LIN {X 0,Y 377.649,Z 370.974,A -85,B 0,C 180,E1 -13185.872,E2 -13185.872} C_VEL
LIN {X 0,Y 374.932,Z 477.201,A -85,B 0,C 180,E1 -13187.993,E2 -13187.993} C_VEL
LIN {X 0,Y 374.183,Z 491.579,A -85,B 0,C 180,E1 -13188.499,E2 -13188.499} C_VEL
LIN {X 0,Y 373.169,Z 505.448,A -85,B 0,C 180,E1 -13189.212,E2 -13189.212} C_VEL
LIN {X 0,Y 372.043,Z 517.617,A -85,B 0,C 180,E1 -13190.04,E2 -13190.04} C_VEL
LIN {X 0,Y 370.513,Z 530.576,A -85,B 0,C 180,E1 -13191.157,E2 -13191.157} C_VEL
LIN {X 0,Y 368.92,Z 542.458,A -85,B 0,C 180,E1 -13192.441,E2 -13192.441} C_VEL
LIN {X 0,Y 367.278,Z 553.835,A -85,B 0,C 180,E1 -13193.957,E2 -13193.957} C_VEL
LIN {X 0,Y 365.706,Z 564.018,A -85,B 0,C 180,E1 -13195.628,E2 -13195.628} C_VEL
LIN {X 0,Y 364.372,Z 572.454,A -85,B 0,C 180,E1 -13197.314,E2 -13197.314} C_VEL
LIN {X 0,Y 363.167,Z 579.995,A -85,B 0,C 180,E1 -13199.149,E2 -13199.149} C_VEL
LIN {X 0,Y 362.222,Z 586.133,A -85,B 0,C 180,E1 -13200.985,E2 -13200.985} C_VEL
LIN {X 0,Y 361.531,Z 591.036,A -85,B 0,C 180,E1 -13202.819,E2 -13202.819} C_VEL
LIN {X 0,Y 361.006,Z 594.853,A -85,B 0,C 180,E1 -13204.642,E2 -13204.642} C_VEL
LIN {X 0,Y 360.671,Z 597.534,A -85,B 0,C 180,E1 -13206.324,E2 -13206.324} C_VEL
LIN {X 0,Y 360.375,Z 599.657,A -85,B 0,C 180,E1 -13208.253,E2 -13208.253} C_VEL
LIN {X 0,Y 360.206,Z 600.871,A -85,B 0,C 180,E1 -13210.63,E2 -13210.63} C_VEL
LIN {X 0,Y 360.181,Z 600.626,A -85,B 0,C 180,E1 -13212.982,E2 -13212.982} C_VEL
LIN {X 0,Y 360.246,Z 598.959,A -85,B 0,C 180,E1 -13215.31,E2 -13215.31} C_VEL
LIN {X 0,Y 360.558,Z 595.855,A -85,B 0,C 180,E1 -13217.62,E2 -13217.62} C_VEL
LIN {X 0,Y 360.942,Z 591.269,A -85,B 0,C 180,E1 -13219.908,E2 -13219.908} C_VEL
LIN {X 0,Y 361.382,Z 586.711,A -85,B 0,C 180,E1 -13221.614,E2 -13221.614} C_VEL
LIN {X 0,Y 362.004,Z 580.162,A -85,B 0,C 180,E1 -13223.592,E2 -13223.592} C_VEL
LIN {X 0,Y 362.969,Z 572.024,A -85,B 0,C 180,E1 -13225.559,E2 -13225.559} C_VEL
LIN {X 0,Y 363.95,Z 563.517,A -85,B 0,C 180,E1 -13227.234,E2 -13227.234} C_VEL
LIN {X 0,Y 365.15,Z 553.229,A -85,B 0,C 180,E1 -13228.898,E2 -13228.898} C_VEL
LIN {X 0,Y 366.336,Z 542.888,A -85,B 0,C 180,E1 -13230.276,E2 -13230.276} C_VEL
LIN {X 0,Y 367.487,Z 531.674,A -85,B 0,C 180,E1 -13231.508,E2 -13231.508} C_VEL
LIN {X 0,Y 368.688,Z 519.413,A -85,B 0,C 180,E1 -13232.596,E2 -13232.596} C_VEL
LIN {X 0,Y 369.825,Z 505.784,A -85,B 0,C 180,E1 -13233.542,E2 -13233.542} C_VEL
LIN {X 0,Y 370.628,Z 491.571,A -85,B 0,C 180,E1 -13234.283,E2 -13234.283} C_VEL
LIN {X 0,Y 371.199,Z 477.507,A -85,B 0,C 180,E1 -13234.786,E2 -13234.786} C_VEL
LIN {X 0,Y 371.887,Z 446.589,A -85,B 0,C 180,E1 -13235.423,E2 -13235.423} C_VEL
LIN {X 0,Y 372.953,Z 396.239,A -85,B 0,C 180,E1 -13236.396,E2 -13236.396} C_VEL
LIN {X 0,Y 372.665,Z 390.402,A -85,B 0,C 180,E1 -13236.533,E2 -13236.533} C_VEL
LIN {X 0,Y 370.599,Z 380.961,A -85,B 0,C 180,E1 -13236.854,E2 -13236.854} C_VEL
LIN {X 0,Y 365.85,Z 366.146,A -85,B 0,C 180,E1 -13237.461,E2 -13237.461} C_VEL
LIN {X 0,Y 357.086,Z 342.727,A -85,B 0,C 180,E1 -13238.539,E2 -13238.539} C_VEL
LIN {X 0,Y 356.134,Z 340.083,A -85,B 0,C 180,E1 -13238.698,E2 -13238.698} C_VEL
LIN {X 0,Y 354.975,Z 334.897,A -85,B 0,C 180,E1 -13240.121,E2 -13240.121} C_VEL
LIN {X 0,Y 354.941,Z 334.894,A -85,B 0,C 180,E1 -13244.02,E2 -13244.02} C_VEL
LIN {X 0,Y 354.889,Z 334.9,A -85,B 0,C 180,E1 -13248.093,E2 -13248.093} C_VEL
LIN {X 0,Y 354.816,Z 334.913,A -85,B 0,C 180,E1 -13251.418,E2 -13251.418} C_VEL
LIN {X 0,Y 354.847,Z 334.907,A -85,B 0,C 180,E1 -13254.578,E2 -13254.578} C_VEL
LIN {X 0,Y 354.796,Z 334.913,A -85,B 0,C 180,E1 -13258.387,E2 -13258.387} C_VEL
LIN {X 0,Y 354.778,Z 334.915,A -85,B 0,C 180,E1 -13262.335,E2 -13262.335} C_VEL
LIN {X 0,Y 354.817,Z 334.909,A -85,B 0,C 180,E1 -13265.699,E2 -13265.699} C_VEL
LIN {X 0,Y 354.768,Z 334.916,A -85,B 0,C 180,E1 -13269.413,E2 -13269.413} C_VEL
LIN {X 0,Y 354.78,Z 334.919,A -85,B 0,C 180,E1 -13272.867,E2 -13272.867} C_VEL
LIN {X 0,Y 354.762,Z 334.916,A -85,B 0,C 180,E1 -13276.104,E2 -13276.104} C_VEL
LIN {X 0,Y 354.763,Z 334.917,A -85,B 0,C 180,E1 -13279.176,E2 -13279.176} C_VEL
LIN {X 0,Y 354.799,Z 334.915,A -85,B 0,C 180,E1 -13282.405,E2 -13282.405} C_VEL
LIN {X 0,Y 354.811,Z 334.912,A -85,B 0,C 180,E1 -13284.941,E2 -13284.941} C_VEL
LIN {X 0,Y 354.795,Z 334.917,A -85,B 0,C 180,E1 -13288.406,E2 -13288.406} C_VEL
LIN {X 0,Y 354.798,Z 334.911,A -85,B 0,C 180,E1 -13291.615,E2 -13291.615} C_VEL
LIN {X 0,Y 354.803,Z 334.911,A -85,B 0,C 180,E1 -13295.42,E2 -13295.42} C_VEL
LIN {X 0,Y 354.824,Z 334.908,A -85,B 0,C 180,E1 -13299.113,E2 -13299.113} C_VEL
LIN {X 0,Y 354.862,Z 334.905,A -85,B 0,C 180,E1 -13302.719,E2 -13302.719} C_VEL
LIN {X 0,Y 354.942,Z 334.899,A -85,B 0,C 180,E1 -13306.255,E2 -13306.255} C_VEL
LIN {X 0,Y 354.959,Z 334.893,A -85,B 0,C 180,E1 -13309.736,E2 -13309.736} C_VEL
LIN {X 0,Y 355.093,Z 334.875,A -85,B 0,C 180,E1 -13313.18,E2 -13313.18} C_VEL
LIN {X 0,Y 355.238,Z 334.86,A -85,B 0,C 180,E1 -13317.733,E2 -13317.733} C_VEL
LIN {X 0,Y 355.334,Z 334.85,A -85,B 0,C 180,E1 -13320,E2 -13320} C_VEL
LIN {X 0,Y 355.236,Z 334.86,A -85,B 0,C 180,E1 -13322.268,E2 -13322.268} C_VEL
LIN {X 0,Y 355.107,Z 334.873,A -85,B 0,C 180,E1 -13326.82,E2 -13326.82} C_VEL
LIN {X 0,Y 354.961,Z 334.893,A -85,B 0,C 180,E1 -13330.265,E2 -13330.265} C_VEL
LIN {X 0,Y 354.947,Z 334.896,A -85,B 0,C 180,E1 -13334.019,E2 -13334.019} C_VEL
LIN {X 0,Y 354.927,Z 334.897,A -85,B 0,C 180,E1 -13338.108,E2 -13338.108} C_VEL
LIN {X 0,Y 354.84,Z 334.908,A -85,B 0,C 180,E1 -13342.106,E2 -13342.106} C_VEL
LIN {X 0,Y 354.904,Z 334.902,A -85,B 0,C 180,E1 -13345.827,E2 -13345.827} C_VEL
LIN {X 0,Y 354.822,Z 334.913,A -85,B 0,C 180,E1 -13349.682,E2 -13349.682} C_VEL
LIN {X 0,Y 354.811,Z 334.913,A -85,B 0,C 180,E1 -13353.702,E2 -13353.702} C_VEL
LIN {X 0,Y 354.804,Z 334.911,A -85,B 0,C 180,E1 -13356.459,E2 -13356.459} C_VEL
LIN {X 0,Y 354.829,Z 334.913,A -85,B 0,C 180,E1 -13359.423,E2 -13359.423} C_VEL
LIN {X 0,Y 354.793,Z 334.914,A -85,B 0,C 180,E1 -13362.867,E2 -13362.867} C_VEL
LIN {X 0,Y 354.785,Z 334.913,A -85,B 0,C 180,E1 -13366.105,E2 -13366.105} C_VEL
LIN {X 0,Y 354.792,Z 334.918,A -85,B 0,C 180,E1 -13369.179,E2 -13369.179} C_VEL
LIN {X 0,Y 354.812,Z 334.91,A -85,B 0,C 180,E1 -13372.402,E2 -13372.402} C_VEL
LIN {X 0,Y 354.817,Z 334.914,A -85,B 0,C 180,E1 -13374.94,E2 -13374.94} C_VEL
LIN {X 0,Y 354.837,Z 334.945,A -85,B 0,C 180,E1 -13376.87,E2 -13376.87} C_VEL
LIN {X 0,Y 357.871,Z 348.237,A -85,B 0,C 180,E1 -13380.042,E2 -13380.042} C_VEL
LIN {X 0,Y 360.045,Z 358.455,A -85,B 0,C 180,E1 -13382.38,E2 -13382.38} C_VEL
LIN {X 0,Y 360.126,Z 361.424,A -85,B 0,C 180,E1 -13383.016,E2 -13383.016} C_VEL
LIN {X 0,Y 359.846,Z 364.189,A -85,B 0,C 180,E1 -13383.584,E2 -13383.584} C_VEL
LIN {X 0,Y 366.367,Z 404.572,A -85,B 0,C 180,E1 -13384.865,E2 -13384.865} C_VEL
LIN {X 0,Y 364.3,Z 502.303,A -85,B 0,C 180,E1 -13386.816,E2 -13386.816} C_VEL
LIN {X 0,Y 363.56,Z 517.056,A -85,B 0,C 180,E1 -13387.33,E2 -13387.33} C_VEL
LIN {X 0,Y 362.525,Z 530.545,A -85,B 0,C 180,E1 -13388.012,E2 -13388.012} C_VEL
LIN {X 0,Y 361.356,Z 543.945,A -85,B 0,C 180,E1 -13388.926,E2 -13388.926} C_VEL
LIN {X 0,Y 360.042,Z 556.534,A -85,B 0,C 180,E1 -13390.025,E2 -13390.025} C_VEL
LIN {X 0,Y 358.731,Z 568.174,A -85,B 0,C 180,E1 -13391.287,E2 -13391.287} C_VEL
LIN {X 0,Y 357.614,Z 577.86,A -85,B 0,C 180,E1 -13392.56,E2 -13392.56} C_VEL
LIN {X 0,Y 356.296,Z 588.612,A -85,B 0,C 180,E1 -13394.262,E2 -13394.262} C_VEL
LIN {X 0,Y 355.379,Z 596.927,A -85,B 0,C 180,E1 -13395.862,E2 -13395.862} C_VEL
LIN {X 0,Y 354.607,Z 604.84,A -85,B 0,C 180,E1 -13397.698,E2 -13397.698} C_VEL
LIN {X 0,Y 353.853,Z 611.86,A -85,B 0,C 180,E1 -13399.702,E2 -13399.702} C_VEL
LIN {X 0,Y 353.555,Z 616.713,A -85,B 0,C 180,E1 -13401.425,E2 -13401.425} C_VEL
LIN {X 0,Y 353.386,Z 620.636,A -85,B 0,C 180,E1 -13403.146,E2 -13403.146} C_VEL
LIN {X 0,Y 353.267,Z 624.452,A -85,B 0,C 180,E1 -13405.435,E2 -13405.435} C_VEL
LIN {X 0,Y 353.239,Z 626.831,A -85,B 0,C 180,E1 -13407.718,E2 -13407.718} C_VEL
LIN {X 0,Y 353.329,Z 627.841,A -85,B 0,C 180,E1 -13409.999,E2 -13409.999} C_VEL
LIN {X 0,Y 353.202,Z 627.494,A -85,B 0,C 180,E1 -13412.28,E2 -13412.28} C_VEL
LIN {X 0,Y 353.247,Z 625.81,A -85,B 0,C 180,E1 -13414.563,E2 -13414.563} C_VEL
LIN {X 0,Y 353.395,Z 622.758,A -85,B 0,C 180,E1 -13416.852,E2 -13416.852} C_VEL
LIN {X 0,Y 353.692,Z 618.263,A -85,B 0,C 180,E1 -13419.146,E2 -13419.146} C_VEL
LIN {X 0,Y 354.128,Z 613.835,A -85,B 0,C 180,E1 -13420.866,E2 -13420.866} C_VEL
LIN {X 0,Y 355.078,Z 607.458,A -85,B 0,C 180,E1 -13422.865,E2 -13422.865} C_VEL
LIN {X 0,Y 356.089,Z 599.558,A -85,B 0,C 180,E1 -13424.866,E2 -13424.866} C_VEL
LIN {X 0,Y 357.377,Z 591.334,A -85,B 0,C 180,E1 -13426.567,E2 -13426.567} C_VEL
LIN {X 0,Y 359,Z 581.461,A -85,B 0,C 180,E1 -13428.253,E2 -13428.253} C_VEL
LIN {X 0,Y 360.756,Z 570.523,A -85,B 0,C 180,E1 -13429.784,E2 -13429.784} C_VEL
LIN {X 0,Y 362.6,Z 558.411,A -85,B 0,C 180,E1 -13431.16,E2 -13431.16} C_VEL
LIN {X 0,Y 364.157,Z 546.5,A -85,B 0,C 180,E1 -13432.255,E2 -13432.255} C_VEL
LIN {X 0,Y 365.623,Z 533.389,A -85,B 0,C 180,E1 -13433.205,E2 -13433.205} C_VEL
LIN {X 0,Y 367.002,Z 519.12,A -85,B 0,C 180,E1 -13433.973,E2 -13433.973} C_VEL
LIN {X 0,Y 368.077,Z 504.919,A -85,B 0,C 180,E1 -13434.499,E2 -13434.499} C_VEL
LIN {X 0,Y 368.736,Z 484.2,A -85,B 0,C 180,E1 -13434.97,E2 -13434.97} C_VEL
LIN {X 0,Y 370.703,Z 405.046,A -85,B 0,C 180,E1 -13436.561,E2 -13436.561} C_VEL
LIN {X 0,Y 366.814,Z 382.746,A -85,B 0,C 180,E1 -13437.423,E2 -13437.423} C_VEL
LIN {X 0,Y 363.097,Z 366.604,A -85,B 0,C 180,E1 -13438.154,E2 -13438.154} C_VEL
LIN {X 0,Y 361.741,Z 363.168,A -85,B 0,C 180,E1 -13438.406,E2 -13438.406} C_VEL
LIN {X 0,Y 359.351,Z 352.096,A -85,B 0,C 180,E1 -13441.214,E2 -13441.214} C_VEL
LIN {X 0,Y 356.366,Z 340.467,A -85,B 0,C 180,E1 -13444.383,E2 -13444.383} C_VEL
LIN {X 0,Y 354.819,Z 334.906,A -85,B 0,C 180,E1 -13446.028,E2 -13446.028} C_VEL
LIN {X 0,Y 354.821,Z 334.908,A -85,B 0,C 180,E1 -13449.422,E2 -13449.422} C_VEL
LIN {X 0,Y 354.8,Z 334.909,A -85,B 0,C 180,E1 -13452.869,E2 -13452.869} C_VEL
LIN {X 0,Y 354.763,Z 334.905,A -85,B 0,C 180,E1 -13456.103,E2 -13456.103} C_VEL
LIN {X 0,Y 354.787,Z 334.909,A -85,B 0,C 180,E1 -13459.178,E2 -13459.178} C_VEL
LIN {X 0,Y 354.807,Z 334.912,A -85,B 0,C 180,E1 -13462.4,E2 -13462.4} C_VEL
LIN {X 0,Y 354.807,Z 334.913,A -85,B 0,C 180,E1 -13464.94,E2 -13464.94} C_VEL
LIN {X 0,Y 354.788,Z 334.917,A -85,B 0,C 180,E1 -13468.404,E2 -13468.404} C_VEL
LIN {X 0,Y 354.848,Z 334.907,A -85,B 0,C 180,E1 -13471.618,E2 -13471.618} C_VEL
LIN {X 0,Y 354.892,Z 334.898,A -85,B 0,C 180,E1 -13474.172,E2 -13474.172} C_VEL
LIN {X 0,Y 354.825,Z 334.905,A -85,B 0,C 180,E1 -13477.893,E2 -13477.893} C_VEL
LIN {X 0,Y 354.915,Z 334.895,A -85,B 0,C 180,E1 -13481.891,E2 -13481.891} C_VEL
LIN {X 0,Y 354.935,Z 334.894,A -85,B 0,C 180,E1 -13485.98,E2 -13485.98} C_VEL
LIN {X 0,Y 354.969,Z 334.887,A -85,B 0,C 180,E1 -13489.735,E2 -13489.735} C_VEL
LIN {X 0,Y 355.105,Z 334.872,A -85,B 0,C 180,E1 -13492.036,E2 -13492.036} C_VEL
LIN {X 0,Y 355.079,Z 334.88,A -85,B 0,C 180,E1 -13494.32,E2 -13494.32} C_VEL
LIN {X 0,Y 355.221,Z 334.856,A -85,B 0,C 180,E1 -13497.732,E2 -13497.732} C_VEL
LIN {X 0,Y 355.136,Z 334.866,A -85,B 0,C 180,E1 -13501.134,E2 -13501.134} C_VEL
LIN {X 0,Y 355.223,Z 334.861,A -85,B 0,C 180,E1 -13502.267,E2 -13502.267} C_VEL
LIN {X 0,Y 355.073,Z 334.879,A -85,B 0,C 180,E1 -13506.82,E2 -13506.82} C_VEL
LIN {X 0,Y 354.944,Z 334.896,A -85,B 0,C 180,E1 -13510.265,E2 -13510.265} C_VEL
LIN {X 0,Y 354.933,Z 334.898,A -85,B 0,C 180,E1 -13514.018,E2 -13514.018} C_VEL
LIN {X 0,Y 354.88,Z 334.903,A -85,B 0,C 180,E1 -13518.092,E2 -13518.092} C_VEL
LIN {X 0,Y 354.806,Z 334.908,A -85,B 0,C 180,E1 -13522.107,E2 -13522.107} C_VEL
LIN {X 0,Y 354.839,Z 334.909,A -85,B 0,C 180,E1 -13524.577,E2 -13524.577} C_VEL
LIN {X 0,Y 354.79,Z 334.902,A -85,B 0,C 180,E1 -13528.386,E2 -13528.386} C_VEL
LIN {X 0,Y 354.778,Z 334.913,A -85,B 0,C 180,E1 -13532.334,E2 -13532.334} C_VEL
LIN {X 0,Y 354.813,Z 334.914,A -85,B 0,C 180,E1 -13535.7,E2 -13535.7} C_VEL
LIN {X 0,Y 354.816,Z 334.906,A -85,B 0,C 180,E1 -13539.424,E2 -13539.424} C_VEL
LIN {X 0,Y 354.803,Z 335.09,A -85,B 0,C 180,E1 -13541.176,E2 -13541.176} C_VEL
LIN {X 0,Y 356.505,Z 341.345,A -85,B 0,C 180,E1 -13543.134,E2 -13543.134} C_VEL
LIN {X 0,Y 366.3,Z 360.999,A -85,B 0,C 180,E1 -13544.598,E2 -13544.598} C_VEL
LIN {X 0,Y 371.482,Z 372.961,A -85,B 0,C 180,E1 -13545.359,E2 -13545.359} C_VEL
LIN {X 0,Y 368.723,Z 476.994,A -85,B 0,C 180,E1 -13547.466,E2 -13547.466} C_VEL
LIN {X 0,Y 367.99,Z 491.14,A -85,B 0,C 180,E1 -13547.963,E2 -13547.963} C_VEL
LIN {X 0,Y 366.946,Z 504.304,A -85,B 0,C 180,E1 -13548.628,E2 -13548.628} C_VEL
LIN {X 0,Y 365.644,Z 517.9,A -85,B 0,C 180,E1 -13549.558,E2 -13549.558} C_VEL
LIN {X 0,Y 364.099,Z 530.421,A -85,B 0,C 180,E1 -13550.65,E2 -13550.65} C_VEL
LIN {X 0,Y 362.576,Z 541.429,A -85,B 0,C 180,E1 -13551.843,E2 -13551.843} C_VEL
LIN {X 0,Y 360.792,Z 553.001,A -85,B 0,C 180,E1 -13553.378,E2 -13553.378} C_VEL
LIN {X 0,Y 359.121,Z 563.612,A -85,B 0,C 180,E1 -13555.117,E2 -13555.117} C_VEL
LIN {X 0,Y 357.576,Z 572.703,A -85,B 0,C 180,E1 -13556.949,E2 -13556.949} C_VEL
LIN {X 0,Y 356.31,Z 580.25,A -85,B 0,C 180,E1 -13558.819,E2 -13558.819} C_VEL
LIN {X 0,Y 355.391,Z 585.721,A -85,B 0,C 180,E1 -13560.471,E2 -13560.471} C_VEL
LIN {X 0,Y 354.648,Z 590.535,A -85,B 0,C 180,E1 -13562.246,E2 -13562.246} C_VEL
LIN {X 0,Y 353.9,Z 595.679,A -85,B 0,C 180,E1 -13564.726,E2 -13564.726} C_VEL
LIN {X 0,Y 353.531,Z 598.345,A -85,B 0,C 180,E1 -13566.574,E2 -13566.574} C_VEL
LIN {X 0,Y 353.205,Z 600.546,A -85,B 0,C 180,E1 -13569.014,E2 -13569.014} C_VEL
LIN {X 0,Y 353.083,Z 601.243,A -85,B 0,C 180,E1 -13571.431,E2 -13571.431} C_VEL
LIN {X 0,Y 353.113,Z 600.455,A -85,B 0,C 180,E1 -13573.822,E2 -13573.822} C_VEL
LIN {X 0,Y 353.218,Z 598.249,A -85,B 0,C 180,E1 -13576.188,E2 -13576.188} C_VEL
LIN {X 0,Y 353.507,Z 595.671,A -85,B 0,C 180,E1 -13577.952,E2 -13577.952} C_VEL
LIN {X 0,Y 353.802,Z 592.19,A -85,B 0,C 180,E1 -13579.703,E2 -13579.703} C_VEL
LIN {X 0,Y 354.242,Z 587.817,A -85,B 0,C 180,E1 -13581.444,E2 -13581.444} C_VEL
LIN {X 0,Y 354.882,Z 581.464,A -85,B 0,C 180,E1 -13583.463,E2 -13583.463} C_VEL
LIN {X 0,Y 355.821,Z 573.552,A -85,B 0,C 180,E1 -13585.47,E2 -13585.47} C_VEL
LIN {X 0,Y 356.793,Z 565.299,A -85,B 0,C 180,E1 -13587.178,E2 -13587.178} C_VEL
LIN {X 0,Y 358.063,Z 555.338,A -85,B 0,C 180,E1 -13588.876,E2 -13588.876} C_VEL
LIN {X 0,Y 359.377,Z 544.282,A -85,B 0,C 180,E1 -13590.421,E2 -13590.421} C_VEL
LIN {X 0,Y 360.536,Z 533.314,A -85,B 0,C 180,E1 -13591.677,E2 -13591.677} C_VEL
LIN {X 0,Y 361.767,Z 521.402,A -85,B 0,C 180,E1 -13592.785,E2 -13592.785} C_VEL
LIN {X 0,Y 362.933,Z 508.295,A -85,B 0,C 180,E1 -13593.748,E2 -13593.748} C_VEL
LIN {X 0,Y 363.798,Z 494.108,A -85,B 0,C 180,E1 -13594.537,E2 -13594.537} C_VEL
LIN {X 0,Y 364.424,Z 481.109,A -85,B 0,C 180,E1 -13595.049,E2 -13595.049} C_VEL
LIN {X 0,Y 364.92,Z 464.085,A -85,B 0,C 180,E1 -13595.458,E2 -13595.458} C_VEL
LIN {X 0,Y 366.898,Z 370.233,A -85,B 0,C 180,E1 -13597.308,E2 -13597.308} C_VEL
LIN {X 0,Y 365.85,Z 366.146,A -85,B 0,C 180,E1 -13597.461,E2 -13597.461} C_VEL
LIN {X 0,Y 363.54,Z 360.985,A -85,B 0,C 180,E1 -13597.72,E2 -13597.72} C_VEL
LIN {X 0,Y 360.254,Z 356.432,A -85,B 0,C 180,E1 -13598.032,E2 -13598.032} C_VEL
LIN {X 0,Y 351.868,Z 346.34,A -85,B 0,C 180,E1 -13598.818,E2 -13598.818} C_VEL
LIN {X 0,Y 349.207,Z 341.334,A -85,B 0,C 180,E1 -13599.117,E2 -13599.117} C_VEL
LIN {X 0,Y 348.965,Z 340.469,A -85,B 0,C 180,E1 -13599.161,E2 -13599.161} C_VEL
LIN {X 0,Y 347.894,Z 335.778,A -85,B 0,C 180,E1 -13600.476,E2 -13600.476} C_VEL
LIN {X 0,Y 347.897,Z 335.772,A -85,B 0,C 180,E1 -13604.151,E2 -13604.151} C_VEL
LIN {X 0,Y 347.828,Z 335.78,A -85,B 0,C 180,E1 -13608.26,E2 -13608.26} C_VEL
LIN {X 0,Y 347.763,Z 335.79,A -85,B 0,C 180,E1 -13611.626,E2 -13611.626} C_VEL
LIN {X 0,Y 347.766,Z 335.794,A -85,B 0,C 180,E1 -13615.113,E2 -13615.113} C_VEL
LIN {X 0,Y 347.743,Z 335.796,A -85,B 0,C 180,E1 -13619.017,E2 -13619.017} C_VEL
LIN {X 0,Y 347.73,Z 335.797,A -85,B 0,C 180,E1 -13623.073,E2 -13623.073} C_VEL
LIN {X 0,Y 347.765,Z 335.787,A -85,B 0,C 180,E1 -13626.065,E2 -13626.065} C_VEL
LIN {X 0,Y 347.73,Z 335.797,A -85,B 0,C 180,E1 -13628.796,E2 -13628.796} C_VEL
LIN {X 0,Y 347.739,Z 335.79,A -85,B 0,C 180,E1 -13631.833,E2 -13631.833} C_VEL
LIN {X 0,Y 347.7,Z 335.798,A -85,B 0,C 180,E1 -13635.029,E2 -13635.029} C_VEL
LIN {X 0,Y 347.738,Z 335.794,A -85,B 0,C 180,E1 -13638.401,E2 -13638.401} C_VEL
LIN {X 0,Y 347.762,Z 335.788,A -85,B 0,C 180,E1 -13642.015,E2 -13642.015} C_VEL
LIN {X 0,Y 347.745,Z 335.789,A -85,B 0,C 180,E1 -13645.537,E2 -13645.537} C_VEL
LIN {X 0,Y 347.746,Z 335.793,A -85,B 0,C 180,E1 -13648.301,E2 -13648.301} C_VEL
LIN {X 0,Y 347.745,Z 335.791,A -85,B 0,C 180,E1 -13650.985,E2 -13650.985} C_VEL
LIN {X 0,Y 347.734,Z 335.791,A -85,B 0,C 180,E1 -13653.6,E2 -13653.6} C_VEL
LIN {X 0,Y 347.75,Z 335.793,A -85,B 0,C 180,E1 -13656.16,E2 -13656.16} C_VEL
LIN {X 0,Y 347.778,Z 335.788,A -85,B 0,C 180,E1 -13659.908,E2 -13659.908} C_VEL
LIN {X 0,Y 347.803,Z 335.783,A -85,B 0,C 180,E1 -13663.567,E2 -13663.567} C_VEL
LIN {X 0,Y 347.89,Z 335.769,A -85,B 0,C 180,E1 -13667.161,E2 -13667.161} C_VEL
LIN {X 0,Y 347.938,Z 335.767,A -85,B 0,C 180,E1 -13670.701,E2 -13670.701} C_VEL
LIN {X 0,Y 348.047,Z 335.757,A -85,B 0,C 180,E1 -13674.206,E2 -13674.206} C_VEL
LIN {X 0,Y 348.199,Z 335.735,A -85,B 0,C 180,E1 -13677.687,E2 -13677.687} C_VEL
LIN {X 0,Y 348.286,Z 335.726,A -85,B 0,C 180,E1 -13680,E2 -13680} C_VEL
LIN {X 0,Y 348.198,Z 335.736,A -85,B 0,C 180,E1 -13682.314,E2 -13682.314} C_VEL
LIN {X 0,Y 348.074,Z 335.749,A -85,B 0,C 180,E1 -13686.959,E2 -13686.959} C_VEL
LIN {X 0,Y 347.901,Z 335.771,A -85,B 0,C 180,E1 -13690.476,E2 -13690.476} C_VEL
LIN {X 0,Y 347.903,Z 335.772,A -85,B 0,C 180,E1 -13694.15,E2 -13694.15} C_VEL
LIN {X 0,Y 347.895,Z 335.772,A -85,B 0,C 180,E1 -13698.29,E2 -13698.29} C_VEL
LIN {X 0,Y 347.795,Z 335.79,A -85,B 0,C 180,E1 -13701.636,E2 -13701.636} C_VEL
LIN {X 0,Y 347.817,Z 335.782,A -85,B 0,C 180,E1 -13705.108,E2 -13705.108} C_VEL
LIN {X 0,Y 347.813,Z 335.786,A -85,B 0,C 180,E1 -13707.694,E2 -13707.694} C_VEL
LIN {X 0,Y 347.754,Z 335.789,A -85,B 0,C 180,E1 -13710.348,E2 -13710.348} C_VEL
LIN {X 0,Y 347.753,Z 335.79,A -85,B 0,C 180,E1 -13714.044,E2 -13714.044} C_VEL
LIN {X 0,Y 347.769,Z 335.793,A -85,B 0,C 180,E1 -13717.32,E2 -13717.32} C_VEL
LIN {X 0,Y 347.737,Z 335.791,A -85,B 0,C 180,E1 -13720.297,E2 -13720.297} C_VEL
LIN {X 0,Y 347.728,Z 335.797,A -85,B 0,C 180,E1 -13723.408,E2 -13723.408} C_VEL
LIN {X 0,Y 347.732,Z 335.793,A -85,B 0,C 180,E1 -13726.685,E2 -13726.685} C_VEL
LIN {X 0,Y 347.751,Z 335.79,A -85,B 0,C 180,E1 -13730.173,E2 -13730.173} C_VEL
LIN {X 0,Y 347.766,Z 335.79,A -85,B 0,C 180,E1 -13732.679,E2 -13732.679} C_VEL
LIN {X 0,Y 347.787,Z 335.786,A -85,B 0,C 180,E1 -13736.445,E2 -13736.445} C_VEL
LIN {X 0,Y 351.046,Z 350.09,A -85,B 0,C 180,E1 -13739.966,E2 -13739.966} C_VEL
LIN {X 0,Y 353.233,Z 360.748,A -85,B 0,C 180,E1 -13742.445,E2 -13742.445} C_VEL
LIN {X 0,Y 353.094,Z 363.95,A -85,B 0,C 180,E1 -13743.127,E2 -13743.127} C_VEL
LIN {X 0,Y 359.723,Z 405.351,A -85,B 0,C 180,E1 -13744.469,E2 -13744.469} C_VEL
LIN {X 0,Y 357.635,Z 502.009,A -85,B 0,C 180,E1 -13746.435,E2 -13746.435} C_VEL
LIN {X 0,Y 356.868,Z 516.772,A -85,B 0,C 180,E1 -13746.957,E2 -13746.957} C_VEL
LIN {X 0,Y 355.807,Z 530.266,A -85,B 0,C 180,E1 -13747.651,E2 -13747.651} C_VEL
LIN {X 0,Y 354.558,Z 543.932,A -85,B 0,C 180,E1 -13748.602,E2 -13748.602} C_VEL
LIN {X 0,Y 353.335,Z 555.54,A -85,B 0,C 180,E1 -13749.629,E2 -13749.629} C_VEL
LIN {X 0,Y 351.911,Z 567.301,A -85,B 0,C 180,E1 -13750.911,E2 -13750.911} C_VEL
LIN {X 0,Y 350.741,Z 577.088,A -85,B 0,C 180,E1 -13752.206,E2 -13752.206} C_VEL
LIN {X 0,Y 349.393,Z 587.927,A -85,B 0,C 180,E1 -13753.943,E2 -13753.943} C_VEL
LIN {X 0,Y 348.32,Z 597.086,A -85,B 0,C 180,E1 -13755.737,E2 -13755.737} C_VEL
LIN {X 0,Y 347.485,Z 605.424,A -85,B 0,C 180,E1 -13757.738,E2 -13757.738} C_VEL
LIN {X 0,Y 346.807,Z 611.367,A -85,B 0,C 180,E1 -13759.49,E2 -13759.49} C_VEL
LIN {X 0,Y 346.486,Z 616.271,A -85,B 0,C 180,E1 -13761.249,E2 -13761.249} C_VEL
LIN {X 0,Y 346.308,Z 620.24,A -85,B 0,C 180,E1 -13763.005,E2 -13763.005} C_VEL
LIN {X 0,Y 346.186,Z 624.099,A -85,B 0,C 180,E1 -13765.341,E2 -13765.341} C_VEL
LIN {X 0,Y 346.145,Z 626.515,A -85,B 0,C 180,E1 -13767.672,E2 -13767.672} C_VEL
LIN {X 0,Y 346.234,Z 627.562,A -85,B 0,C 180,E1 -13769.999,E2 -13769.999} C_VEL
LIN {X 0,Y 346.111,Z 627.252,A -85,B 0,C 180,E1 -13772.326,E2 -13772.326} C_VEL
LIN {X 0,Y 346.146,Z 625.607,A -85,B 0,C 180,E1 -13774.657,E2 -13774.657} C_VEL
LIN {X 0,Y 346.32,Z 622.596,A -85,B 0,C 180,E1 -13776.993,E2 -13776.993} C_VEL
LIN {X 0,Y 346.648,Z 618.142,A -85,B 0,C 180,E1 -13779.333,E2 -13779.333} C_VEL
LIN {X 0,Y 347.352,Z 612.126,A -85,B 0,C 180,E1 -13781.672,E2 -13781.672} C_VEL
LIN {X 0,Y 348.334,Z 605.389,A -85,B 0,C 180,E1 -13783.712,E2 -13783.712} C_VEL
LIN {X 0,Y 349.635,Z 597.041,A -85,B 0,C 180,E1 -13785.744,E2 -13785.744} C_VEL
LIN {X 0,Y 351.077,Z 588.387,A -85,B 0,C 180,E1 -13787.473,E2 -13787.473} C_VEL
LIN {X 0,Y 352.891,Z 577.94,A -85,B 0,C 180,E1 -13789.183,E2 -13789.183} C_VEL
LIN {X 0,Y 354.809,Z 566.292,A -85,B 0,C 180,E1 -13790.735,E2 -13790.735} C_VEL
LIN {X 0,Y 356.549,Z 554.676,A -85,B 0,C 180,E1 -13791.993,E2 -13791.993} C_VEL
LIN {X 0,Y 358.248,Z 541.93,A -85,B 0,C 180,E1 -13793.1,E2 -13793.1} C_VEL
LIN {X 0,Y 359.782,Z 528.732,A -85,B 0,C 180,E1 -13793.987,E2 -13793.987} C_VEL
LIN {X 0,Y 361.083,Z 515.203,A -85,B 0,C 180,E1 -13794.66,E2 -13794.66} C_VEL
LIN {X 0,Y 362.01,Z 501.478,A -85,B 0,C 180,E1 -13795.129,E2 -13795.129} C_VEL
LIN {X 0,Y 364.561,Z 406.286,A -85,B 0,C 180,E1 -13797.095,E2 -13797.095} C_VEL
LIN {X 0,Y 360.933,Z 384.935,A -85,B 0,C 180,E1 -13797.94,E2 -13797.94} C_VEL
LIN {X 0,Y 357.328,Z 369.42,A -85,B 0,C 180,E1 -13798.672,E2 -13798.672} C_VEL
LIN {X 0,Y 354.555,Z 362.91,A -85,B 0,C 180,E1 -13799.139,E2 -13799.139} C_VEL
LIN {X 0,Y 351.838,Z 350.947,A -85,B 0,C 180,E1 -13802.297,E2 -13802.297} C_VEL
LIN {X 0,Y 349.331,Z 341.44,A -85,B 0,C 180,E1 -13804.993,E2 -13804.993} C_VEL
LIN {X 0,Y 347.772,Z 335.786,A -85,B 0,C 180,E1 -13806.724,E2 -13806.724} C_VEL
LIN {X 0,Y 347.752,Z 335.796,A -85,B 0,C 180,E1 -13810.293,E2 -13810.293} C_VEL
LIN {X 0,Y 347.74,Z 335.796,A -85,B 0,C 180,E1 -13813.404,E2 -13813.404} C_VEL
LIN {X 0,Y 347.721,Z 335.786,A -85,B 0,C 180,E1 -13816.685,E2 -13816.685} C_VEL
LIN {X 0,Y 347.743,Z 335.776,A -85,B 0,C 180,E1 -13820.172,E2 -13820.172} C_VEL
LIN {X 0,Y 347.76,Z 335.794,A -85,B 0,C 180,E1 -13822.679,E2 -13822.679} C_VEL
LIN {X 0,Y 347.742,Z 335.795,A -85,B 0,C 180,E1 -13825.955,E2 -13825.955} C_VEL
LIN {X 0,Y 347.758,Z 335.79,A -85,B 0,C 180,E1 -13829.653,E2 -13829.653} C_VEL
LIN {X 0,Y 347.846,Z 335.777,A -85,B 0,C 180,E1 -13832.743,E2 -13832.743} C_VEL
LIN {X 0,Y 347.779,Z 335.787,A -85,B 0,C 180,E1 -13836.161,E2 -13836.161} C_VEL
LIN {X 0,Y 347.805,Z 335.784,A -85,B 0,C 180,E1 -13839.909,E2 -13839.909} C_VEL
LIN {X 0,Y 347.859,Z 335.78,A -85,B 0,C 180,E1 -13842.359,E2 -13842.359} C_VEL
LIN {X 0,Y 347.89,Z 335.771,A -85,B 0,C 180,E1 -13845.97,E2 -13845.97} C_VEL
LIN {X 0,Y 347.92,Z 335.763,A -85,B 0,C 180,E1 -13849.525,E2 -13849.525} C_VEL
LIN {X 0,Y 348.065,Z 335.751,A -85,B 0,C 180,E1 -13851.874,E2 -13851.874} C_VEL
LIN {X 0,Y 348.055,Z 335.753,A -85,B 0,C 180,E1 -13854.205,E2 -13854.205} C_VEL
LIN {X 0,Y 348.183,Z 335.732,A -85,B 0,C 180,E1 -13857.686,E2 -13857.686} C_VEL
LIN {X 0,Y 348.107,Z 335.741,A -85,B 0,C 180,E1 -13861.156,E2 -13861.156} C_VEL
LIN {X 0,Y 348.185,Z 335.737,A -85,B 0,C 180,E1 -13862.313,E2 -13862.313} C_VEL
LIN {X 0,Y 348.04,Z 335.755,A -85,B 0,C 180,E1 -13866.959,E2 -13866.959} C_VEL
LIN {X 0,Y 347.884,Z 335.775,A -85,B 0,C 180,E1 -13870.475,E2 -13870.475} C_VEL
LIN {X 0,Y 347.89,Z 335.775,A -85,B 0,C 180,E1 -13874.15,E2 -13874.15} C_VEL
LIN {X 0,Y 347.819,Z 335.783,A -85,B 0,C 180,E1 -13878.259,E2 -13878.259} C_VEL
LIN {X 0,Y 347.758,Z 335.788,A -85,B 0,C 180,E1 -13881.626,E2 -13881.626} C_VEL
LIN {X 0,Y 347.759,Z 335.79,A -85,B 0,C 180,E1 -13885.112,E2 -13885.112} C_VEL
LIN {X 0,Y 347.727,Z 335.787,A -85,B 0,C 180,E1 -13887.701,E2 -13887.701} C_VEL
LIN {X 0,Y 347.732,Z 335.798,A -85,B 0,C 180,E1 -13890.349,E2 -13890.349} C_VEL
LIN {X 0,Y 347.74,Z 335.793,A -85,B 0,C 180,E1 -13894.044,E2 -13894.044} C_VEL
LIN {X 0,Y 347.752,Z 335.789,A -85,B 0,C 180,E1 -13897.321,E2 -13897.321} C_VEL
LIN {X 0,Y 347.757,Z 335.873,A -85,B 0,C 180,E1 -13900.483,E2 -13900.483} C_VEL
LIN {X 0,Y 349.262,Z 341.566,A -85,B 0,C 180,E1 -13902.343,E2 -13902.343} C_VEL
LIN {X 0,Y 359.506,Z 361.601,A -85,B 0,C 180,E1 -13903.934,E2 -13903.934} C_VEL
LIN {X 0,Y 365.379,Z 374.94,A -85,B 0,C 180,E1 -13904.83,E2 -13904.83} C_VEL
LIN {X 0,Y 362.51,Z 477.449,A -85,B 0,C 180,E1 -13906.94,E2 -13906.94} C_VEL
LIN {X 0,Y 361.734,Z 491.51,A -85,B 0,C 180,E1 -13907.442,E2 -13907.442} C_VEL
LIN {X 0,Y 360.65,Z 504.591,A -85,B 0,C 180,E1 -13908.113,E2 -13908.113} C_VEL
LIN {X 0,Y 359.276,Z 518.218,A -85,B 0,C 180,E1 -13909.058,E2 -13909.058} C_VEL
LIN {X 0,Y 357.741,Z 530.294,A -85,B 0,C 180,E1 -13910.126,E2 -13910.126} C_VEL
LIN {X 0,Y 356.075,Z 541.729,A -85,B 0,C 180,E1 -13911.379,E2 -13911.379} C_VEL
LIN {X 0,Y 354.341,Z 552.595,A -85,B 0,C 180,E1 -13912.838,E2 -13912.838} C_VEL
LIN {X 0,Y 352.768,Z 561.938,A -85,B 0,C 180,E1 -13914.359,E2 -13914.359} C_VEL
LIN {X 0,Y 351.063,Z 571.519,A -85,B 0,C 180,E1 -13916.254,E2 -13916.254} C_VEL
LIN {X 0,Y 349.798,Z 578.601,A -85,B 0,C 180,E1 -13917.966,E2 -13917.966} C_VEL
LIN {X 0,Y 348.496,Z 585.888,A -85,B 0,C 180,E1 -13920.13,E2 -13920.13} C_VEL
LIN {X 0,Y 347.574,Z 591.556,A -85,B 0,C 180,E1 -13922.287,E2 -13922.287} C_VEL
LIN {X 0,Y 346.966,Z 595.38,A -85,B 0,C 180,E1 -13924.185,E2 -13924.185} C_VEL
LIN {X 0,Y 346.547,Z 598.232,A -85,B 0,C 180,E1 -13926.073,E2 -13926.073} C_VEL
LIN {X 0,Y 346.151,Z 600.61,A -85,B 0,C 180,E1 -13928.565,E2 -13928.565} C_VEL
LIN {X 0,Y 346.015,Z 601.486,A -85,B 0,C 180,E1 -13931.037,E2 -13931.037} C_VEL
LIN {X 0,Y 346.005,Z 600.913,A -85,B 0,C 180,E1 -13933.48,E2 -13933.48} C_VEL
LIN {X 0,Y 346.117,Z 598.895,A -85,B 0,C 180,E1 -13935.898,E2 -13935.898} C_VEL
LIN {X 0,Y 346.492,Z 595.397,A -85,B 0,C 180,E1 -13938.299,E2 -13938.299} C_VEL
LIN {X 0,Y 346.934,Z 590.391,A -85,B 0,C 180,E1 -13940.675,E2 -13940.675} C_VEL
LIN {X 0,Y 347.547,Z 585.148,A -85,B 0,C 180,E1 -13942.573,E2 -13942.573} C_VEL
LIN {X 0,Y 348.239,Z 578.552,A -85,B 0,C 180,E1 -13944.5,E2 -13944.5} C_VEL
LIN {X 0,Y 349.374,Z 569.87,A -85,B 0,C 180,E1 -13946.541,E2 -13946.541} C_VEL
LIN {X 0,Y 350.543,Z 560.807,A -85,B 0,C 180,E1 -13948.278,E2 -13948.278} C_VEL
LIN {X 0,Y 351.839,Z 549.87,A -85,B 0,C 180,E1 -13950.001,E2 -13950.001} C_VEL
LIN {X 0,Y 353.222,Z 538.706,A -85,B 0,C 180,E1 -13951.426,E2 -13951.426} C_VEL
LIN {X 0,Y 354.517,Z 526.412,A -85,B 0,C 180,E1 -13952.7,E2 -13952.7} C_VEL
LIN {X 0,Y 355.823,Z 512.609,A -85,B 0,C 180,E1 -13953.823,E2 -13953.823} C_VEL
LIN {X 0,Y 356.831,Z 499.154,A -85,B 0,C 180,E1 -13954.661,E2 -13954.661} C_VEL
LIN {X 0,Y 357.57,Z 485.359,A -85,B 0,C 180,E1 -13955.287,E2 -13955.287} C_VEL
LIN {X 0,Y 358.123,Z 472.492,A -85,B 0,C 180,E1 -13955.667,E2 -13955.667} C_VEL
LIN {X 0,Y 360.314,Z 371.491,A -85,B 0,C 180,E1 -13957.704,E2 -13957.704} C_VEL
LIN {X 0,Y 358.222,Z 364.76,A -85,B 0,C 180,E1 -13957.985,E2 -13957.985} C_VEL
LIN {X 0,Y 349.894,Z 342.978,A -85,B 0,C 180,E1 -13959.031,E2 -13959.031} C_VEL
LIN {X 0,Y 349.207,Z 341.334,A -85,B 0,C 180,E1 -13959.117,E2 -13959.117} C_VEL
LIN {X 0,Y 348.09,Z 340.136,A -85,B 0,C 180,E1 -13959.316,E2 -13959.316} C_VEL
LIN {X 0,Y 343.923,Z 337.36,A -85,B 0,C 180,E1 -13960.411,E2 -13960.411} C_VEL
LIN {X 0,Y 341.407,Z 336.789,A -85,B 0,C 180,E1 -13961.523,E2 -13961.523} C_VEL
LIN {X 0,Y 340.83,Z 336.652,A -85,B 0,C 180,E1 -13962.267,E2 -13962.267} C_VEL
LIN {X 0,Y 340.816,Z 336.657,A -85,B 0,C 180,E1 -13965.551,E2 -13965.551} C_VEL
LIN {X 0,Y 340.762,Z 336.666,A -85,B 0,C 180,E1 -13969.269,E2 -13969.269} C_VEL
LIN {X 0,Y 340.705,Z 336.673,A -85,B 0,C 180,E1 -13973.075,E2 -13973.075} C_VEL
LIN {X 0,Y 340.714,Z 336.667,A -85,B 0,C 180,E1 -13975.67,E2 -13975.67} C_VEL
LIN {X 0,Y 340.701,Z 336.668,A -85,B 0,C 180,E1 -13979.676,E2 -13979.676} C_VEL
LIN {X 0,Y 340.68,Z 336.671,A -85,B 0,C 180,E1 -13982.437,E2 -13982.437} C_VEL
LIN {X 0,Y 340.715,Z 336.667,A -85,B 0,C 180,E1 -13985.28,E2 -13985.28} C_VEL
LIN {X 0,Y 340.692,Z 336.669,A -85,B 0,C 180,E1 -13988.383,E2 -13988.383} C_VEL
LIN {X 0,Y 340.69,Z 336.669,A -85,B 0,C 180,E1 -13992.045,E2 -13992.045} C_VEL
LIN {X 0,Y 340.649,Z 336.674,A -85,B 0,C 180,E1 -13996.228,E2 -13996.228} C_VEL
LIN {X 0,Y 340.669,Z 336.677,A -85,B 0,C 180,E1 -13998.689,E2 -13998.689} C_VEL
LIN {X 0,Y 340.718,Z 336.664,A -85,B 0,C 180,E1 -14001.771,E2 -14001.771} C_VEL
LIN {X 0,Y 340.724,Z 336.663,A -85,B 0,C 180,E1 -14005.596,E2 -14005.596} C_VEL
LIN {X 0,Y 340.695,Z 336.67,A -85,B 0,C 180,E1 -14008.956,E2 -14008.956} C_VEL
LIN {X 0,Y 340.711,Z 336.667,A -85,B 0,C 180,E1 -14013.013,E2 -14013.013} C_VEL
LIN {X 0,Y 340.702,Z 336.668,A -85,B 0,C 180,E1 -14016.926,E2 -14016.926} C_VEL
LIN {X 0,Y 340.723,Z 336.667,A -85,B 0,C 180,E1 -14020.73,E2 -14020.73} C_VEL
LIN {X 0,Y 340.796,Z 336.658,A -85,B 0,C 180,E1 -14024.45,E2 -14024.45} C_VEL
LIN {X 0,Y 340.852,Z 336.649,A -85,B 0,C 180,E1 -14028.101,E2 -14028.101} C_VEL
LIN {X 0,Y 340.983,Z 336.634,A -85,B 0,C 180,E1 -14031.705,E2 -14031.705} C_VEL
LIN {X 0,Y 341.021,Z 336.634,A -85,B 0,C 180,E1 -14034.086,E2 -14034.086} C_VEL
LIN {X 0,Y 341.161,Z 336.611,A -85,B 0,C 180,E1 -14037.639,E2 -14037.639} C_VEL
LIN {X 0,Y 341.237,Z 336.602,A -85,B 0,C 180,E1 -14040,E2 -14040} C_VEL
LIN {X 0,Y 341.135,Z 336.615,A -85,B 0,C 180,E1 -14042.362,E2 -14042.362} C_VEL
LIN {X 0,Y 341.022,Z 336.628,A -85,B 0,C 180,E1 -14047.103,E2 -14047.103} C_VEL
LIN {X 0,Y 340.852,Z 336.649,A -85,B 0,C 180,E1 -14050.695,E2 -14050.695} C_VEL
LIN {X 0,Y 340.868,Z 336.647,A -85,B 0,C 180,E1 -14054.325,E2 -14054.325} C_VEL
LIN {X 0,Y 340.842,Z 336.65,A -85,B 0,C 180,E1 -14058.466,E2 -14058.466} C_VEL
LIN {X 0,Y 340.759,Z 336.664,A -85,B 0,C 180,E1 -14061.857,E2 -14061.857} C_VEL
LIN {X 0,Y 340.777,Z 336.663,A -85,B 0,C 180,E1 -14065.664,E2 -14065.664} C_VEL
LIN {X 0,Y 340.733,Z 336.663,A -85,B 0,C 180,E1 -14068.321,E2 -14068.321} C_VEL
LIN {X 0,Y 340.702,Z 336.669,A -85,B 0,C 180,E1 -14071.045,E2 -14071.045} C_VEL
LIN {X 0,Y 340.723,Z 336.67,A -85,B 0,C 180,E1 -14075.279,E2 -14075.279} C_VEL
LIN {X 0,Y 340.716,Z 336.664,A -85,B 0,C 180,E1 -14078.386,E2 -14078.386} C_VEL
LIN {X 0,Y 340.704,Z 336.668,A -85,B 0,C 180,E1 -14082.045,E2 -14082.045} C_VEL
LIN {X 0,Y 340.689,Z 336.673,A -85,B 0,C 180,E1 -14085.461,E2 -14085.461} C_VEL
LIN {X 0,Y 340.69,Z 336.671,A -85,B 0,C 180,E1 -14088.69,E2 -14088.69} C_VEL
LIN {X 0,Y 340.737,Z 336.665,A -85,B 0,C 180,E1 -14091.772,E2 -14091.772} C_VEL
LIN {X 0,Y 340.727,Z 336.667,A -85,B 0,C 180,E1 -14095.595,E2 -14095.595} C_VEL
LIN {X 0,Y 340.712,Z 336.668,A -85,B 0,C 180,E1 -14096.085,E2 -14096.085} C_VEL
LIN {X 0,Y 343.965,Z 350.84,A -85,B 0,C 180,E1 -14099.621,E2 -14099.621} C_VEL
LIN {X 0,Y 346.209,Z 361.512,A -85,B 0,C 180,E1 -14102.166,E2 -14102.166} C_VEL
LIN {X 0,Y 346.338,Z 364.041,A -85,B 0,C 180,E1 -14102.672,E2 -14102.672} C_VEL
LIN {X 0,Y 353.04,Z 405.149,A -85,B 0,C 180,E1 -14104.036,E2 -14104.036} C_VEL
LIN {X 0,Y 351.191,Z 495.684,A -85,B 0,C 180,E1 -14105.897,E2 -14105.897} C_VEL
LIN {X 0,Y 350.55,Z 510.316,A -85,B 0,C 180,E1 -14106.321,E2 -14106.321} C_VEL
LIN {X 0,Y 349.523,Z 525.036,A -85,B 0,C 180,E1 -14106.992,E2 -14106.992} C_VEL
LIN {X 0,Y 348.302,Z 538.514,A -85,B 0,C 180,E1 -14107.847,E2 -14107.847} C_VEL
LIN {X 0,Y 347.037,Z 551.565,A -85,B 0,C 180,E1 -14108.932,E2 -14108.932} C_VEL
LIN {X 0,Y 345.673,Z 562.755,A -85,B 0,C 180,E1 -14110.089,E2 -14110.089} C_VEL
LIN {X 0,Y 344.158,Z 574.295,A -85,B 0,C 180,E1 -14111.546,E2 -14111.546} C_VEL
LIN {X 0,Y 342.904,Z 583.856,A -85,B 0,C 180,E1 -14113.018,E2 -14113.018} C_VEL
LIN {X 0,Y 341.747,Z 593.499,A -85,B 0,C 180,E1 -14114.805,E2 -14114.805} C_VEL
LIN {X 0,Y 340.882,Z 601.42,A -85,B 0,C 180,E1 -14116.588,E2 -14116.588} C_VEL
LIN {X 0,Y 339.993,Z 609.025,A -85,B 0,C 180,E1 -14118.674,E2 -14118.674} C_VEL
LIN {X 0,Y 339.514,Z 614.289,A -85,B 0,C 180,E1 -14120.467,E2 -14120.467} C_VEL
LIN {X 0,Y 339.232,Z 619.827,A -85,B 0,C 180,E1 -14122.858,E2 -14122.858} C_VEL
LIN {X 0,Y 339.088,Z 623.738,A -85,B 0,C 180,E1 -14125.243,E2 -14125.243} C_VEL
LIN {X 0,Y 339.055,Z 626.196,A -85,B 0,C 180,E1 -14127.623,E2 -14127.623} C_VEL
LIN {X 0,Y 339.14,Z 627.282,A -85,B 0,C 180,E1 -14129.999,E2 -14129.999} C_VEL
LIN {X 0,Y 339.023,Z 627.011,A -85,B 0,C 180,E1 -14132.375,E2 -14132.375} C_VEL
LIN {X 0,Y 339.05,Z 625.404,A -85,B 0,C 180,E1 -14134.755,E2 -14134.755} C_VEL
LIN {X 0,Y 339.245,Z 622.432,A -85,B 0,C 180,E1 -14137.139,E2 -14137.139} C_VEL
LIN {X 0,Y 339.618,Z 618.021,A -85,B 0,C 180,E1 -14139.528,E2 -14139.528} C_VEL
LIN {X 0,Y 340.381,Z 612.059,A -85,B 0,C 180,E1 -14141.915,E2 -14141.915} C_VEL
LIN {X 0,Y 341.4,Z 605.388,A -85,B 0,C 180,E1 -14143.997,E2 -14143.997} C_VEL
LIN {X 0,Y 342.758,Z 597.131,A -85,B 0,C 180,E1 -14146.068,E2 -14146.068} C_VEL
LIN {X 0,Y 344.294,Z 588.554,A -85,B 0,C 180,E1 -14147.829,E2 -14147.829} C_VEL
LIN {X 0,Y 346.197,Z 578.193,A -85,B 0,C 180,E1 -14149.569,E2 -14149.569} C_VEL
LIN {X 0,Y 348.198,Z 566.65,A -85,B 0,C 180,E1 -14151.147,E2 -14151.147} C_VEL
LIN {X 0,Y 350.192,Z 553.895,A -85,B 0,C 180,E1 -14152.553,E2 -14152.553} C_VEL
LIN {X 0,Y 351.992,Z 540.852,A -85,B 0,C 180,E1 -14153.691,E2 -14153.691} C_VEL
LIN {X 0,Y 353.636,Z 527.419,A -85,B 0,C 180,E1 -14154.587,E2 -14154.587} C_VEL
LIN {X 0,Y 354.955,Z 513.421,A -85,B 0,C 180,E1 -14155.272,E2 -14155.272} C_VEL
LIN {X 0,Y 355.915,Z 498.667,A -85,B 0,C 180,E1 -14155.747,E2 -14155.747} C_VEL
LIN {X 0,Y 358.486,Z 407.326,A -85,B 0,C 180,E1 -14157.656,E2 -14157.656} C_VEL
LIN {X 0,Y 354.906,Z 386.367,A -85,B 0,C 180,E1 -14158.514,E2 -14158.514} C_VEL
LIN {X 0,Y 351.778,Z 372.601,A -85,B 0,C 180,E1 -14159.177,E2 -14159.177} C_VEL
LIN {X 0,Y 347.351,Z 362.582,A -85,B 0,C 180,E1 -14159.926,E2 -14159.926} C_VEL
LIN {X 0,Y 344.771,Z 351.61,A -85,B 0,C 180,E1 -14162.934,E2 -14162.934} C_VEL
LIN {X 0,Y 342.552,Z 343.103,A -85,B 0,C 180,E1 -14165.42,E2 -14165.42} C_VEL
LIN {X 0,Y 340.73,Z 336.669,A -85,B 0,C 180,E1 -14167.478,E2 -14167.478} C_VEL
LIN {X 0,Y 340.7,Z 336.663,A -85,B 0,C 180,E1 -14171.306,E2 -14171.306} C_VEL
LIN {X 0,Y 340.644,Z 336.674,A -85,B 0,C 180,E1 -14174.543,E2 -14174.543} C_VEL
LIN {X 0,Y 340.695,Z 336.672,A -85,B 0,C 180,E1 -14177.953,E2 -14177.953} C_VEL
LIN {X 0,Y 340.73,Z 336.661,A -85,B 0,C 180,E1 -14181.772,E2 -14181.772} C_VEL
LIN {X 0,Y 340.717,Z 336.668,A -85,B 0,C 180,E1 -14185.594,E2 -14185.594} C_VEL
LIN {X 0,Y 340.698,Z 336.67,A -85,B 0,C 180,E1 -14188.955,E2 -14188.955} C_VEL
LIN {X 0,Y 340.773,Z 336.66,A -85,B 0,C 180,E1 -14192.473,E2 -14192.473} C_VEL
LIN {X 0,Y 340.748,Z 336.665,A -85,B 0,C 180,E1 -14195.637,E2 -14195.637} C_VEL
LIN {X 0,Y 340.738,Z 336.666,A -85,B 0,C 180,E1 -14199.473,E2 -14199.473} C_VEL
LIN {X 0,Y 340.85,Z 336.648,A -85,B 0,C 180,E1 -14201.983,E2 -14201.983} C_VEL
LIN {X 0,Y 340.862,Z 336.644,A -85,B 0,C 180,E1 -14205.704,E2 -14205.704} C_VEL
LIN {X 0,Y 340.862,Z 336.64,A -85,B 0,C 180,E1 -14209.306,E2 -14209.306} C_VEL
LIN {X 0,Y 341.066,Z 336.616,A -85,B 0,C 180,E1 -14212.898,E2 -14212.898} C_VEL
LIN {X 0,Y 341.12,Z 336.611,A -85,B 0,C 180,E1 -14217.638,E2 -14217.638} C_VEL
LIN {X 0,Y 341.079,Z 336.616,A -85,B 0,C 180,E1 -14221.18,E2 -14221.18} C_VEL
LIN {X 0,Y 341.122,Z 336.617,A -85,B 0,C 180,E1 -14222.361,E2 -14222.361} C_VEL
LIN {X 0,Y 340.988,Z 336.635,A -85,B 0,C 180,E1 -14227.103,E2 -14227.103} C_VEL
LIN {X 0,Y 340.836,Z 336.653,A -85,B 0,C 180,E1 -14230.694,E2 -14230.694} C_VEL
LIN {X 0,Y 340.854,Z 336.651,A -85,B 0,C 180,E1 -14234.325,E2 -14234.325} C_VEL
LIN {X 0,Y 340.776,Z 336.66,A -85,B 0,C 180,E1 -14238.44,E2 -14238.44} C_VEL
LIN {X 0,Y 340.709,Z 336.664,A -85,B 0,C 180,E1 -14241.842,E2 -14241.842} C_VEL
LIN {X 0,Y 340.71,Z 336.671,A -85,B 0,C 180,E1 -14245.669,E2 -14245.669} C_VEL
LIN {X 0,Y 340.699,Z 336.663,A -85,B 0,C 180,E1 -14249.674,E2 -14249.674} C_VEL
LIN {X 0,Y 340.677,Z 336.668,A -85,B 0,C 180,E1 -14252.436,E2 -14252.436} C_VEL
LIN {X 0,Y 340.709,Z 336.674,A -85,B 0,C 180,E1 -14255.279,E2 -14255.279} C_VEL
LIN {X 0,Y 340.7,Z 336.666,A -85,B 0,C 180,E1 -14259.016,E2 -14259.016} C_VEL
LIN {X 0,Y 340.701,Z 336.676,A -85,B 0,C 180,E1 -14259.752,E2 -14259.752} C_VEL
LIN {X 0,Y 342.148,Z 342.021,A -85,B 0,C 180,E1 -14261.536,E2 -14261.536} C_VEL
LIN {X 0,Y 346.372,Z 349.762,A -85,B 0,C 180,E1 -14262.228,E2 -14262.228} C_VEL
LIN {X 0,Y 355.334,Z 367.82,A -85,B 0,C 180,E1 -14263.652,E2 -14263.652} C_VEL
LIN {X 0,Y 359.295,Z 377.236,A -85,B 0,C 180,E1 -14264.283,E2 -14264.283} C_VEL
LIN {X 0,Y 356.345,Z 477.628,A -85,B 0,C 180,E1 -14266.383,E2 -14266.383} C_VEL
LIN {X 0,Y 355.535,Z 491.831,A -85,B 0,C 180,E1 -14266.899,E2 -14266.899} C_VEL
LIN {X 0,Y 354.368,Z 505.239,A -85,B 0,C 180,E1 -14267.602,E2 -14267.602} C_VEL
LIN {X 0,Y 352.946,Z 518.546,A -85,B 0,C 180,E1 -14268.543,E2 -14268.543} C_VEL
LIN {X 0,Y 351.216,Z 531.44,A -85,B 0,C 180,E1 -14269.71,E2 -14269.71} C_VEL
LIN {X 0,Y 349.383,Z 543.303,A -85,B 0,C 180,E1 -14271.054,E2 -14271.054} C_VEL
LIN {X 0,Y 347.472,Z 554.651,A -85,B 0,C 180,E1 -14272.644,E2 -14272.644} C_VEL
LIN {X 0,Y 345.639,Z 564.916,A -85,B 0,C 180,E1 -14274.422,E2 -14274.422} C_VEL
LIN {X 0,Y 344.068,Z 573.249,A -85,B 0,C 180,E1 -14276.18,E2 -14276.18} C_VEL
LIN {X 0,Y 342.647,Z 580.789,A -85,B 0,C 180,E1 -14278.121,E2 -14278.121} C_VEL
LIN {X 0,Y 341.322,Z 587.795,A -85,B 0,C 180,E1 -14280.386,E2 -14280.386} C_VEL
LIN {X 0,Y 340.381,Z 593.102,A -85,B 0,C 180,E1 -14282.602,E2 -14282.602} C_VEL
LIN {X 0,Y 339.864,Z 596.21,A -85,B 0,C 180,E1 -14284.263,E2 -14284.263} C_VEL
LIN {X 0,Y 339.563,Z 598.177,A -85,B 0,C 180,E1 -14285.598,E2 -14285.598} C_VEL
LIN {X 0,Y 339.109,Z 600.674,A -85,B 0,C 180,E1 -14288.098,E2 -14288.098} C_VEL
LIN {X 0,Y 338.92,Z 601.72,A -85,B 0,C 180,E1 -14290.624,E2 -14290.624} C_VEL
LIN {X 0,Y 338.915,Z 601.312,A -85,B 0,C 180,E1 -14293.124,E2 -14293.124} C_VEL
LIN {X 0,Y 338.99,Z 599.486,A -85,B 0,C 180,E1 -14295.596,E2 -14295.596} C_VEL
LIN {X 0,Y 339.339,Z 596.212,A -85,B 0,C 180,E1 -14298.048,E2 -14298.048} C_VEL
LIN {X 0,Y 339.801,Z 591.385,A -85,B 0,C 180,E1 -14300.477,E2 -14300.477} C_VEL
LIN {X 0,Y 340.39,Z 586.604,A -85,B 0,C 180,E1 -14302.325,E2 -14302.325} C_VEL
LIN {X 0,Y 341.089,Z 579.949,A -85,B 0,C 180,E1 -14304.384,E2 -14304.384} C_VEL
LIN {X 0,Y 342.213,Z 571.507,A -85,B 0,C 180,E1 -14306.469,E2 -14306.469} C_VEL
LIN {X 0,Y 343.385,Z 562.716,A -85,B 0,C 180,E1 -14308.242,E2 -14308.242} C_VEL
LIN {X 0,Y 344.74,Z 552.082,A -85,B 0,C 180,E1 -14310.001,E2 -14310.001} C_VEL
LIN {X 0,Y 346.106,Z 541.324,A -85,B 0,C 180,E1 -14311.455,E2 -14311.455} C_VEL
LIN {X 0,Y 347.442,Z 529.584,A -85,B 0,C 180,E1 -14312.755,E2 -14312.755} C_VEL
LIN {X 0,Y 348.745,Z 516.656,A -85,B 0,C 180,E1 -14313.901,E2 -14313.901} C_VEL
LIN {X 0,Y 349.858,Z 503.197,A -85,B 0,C 180,E1 -14314.826,E2 -14314.826} C_VEL
LIN {X 0,Y 350.69,Z 489.167,A -85,B 0,C 180,E1 -14315.535,E2 -14315.535} C_VEL
LIN {X 0,Y 351.343,Z 475.588,A -85,B 0,C 180,E1 -14315.993,E2 -14315.993} C_VEL
LIN {X 0,Y 353.653,Z 372.066,A -85,B 0,C 180,E1 -14318.129,E2 -14318.129} C_VEL
LIN {X 0,Y 344.798,Z 348.263,A -85,B 0,C 180,E1 -14319.277,E2 -14319.277} C_VEL
LIN {X 0,Y 341.736,Z 340.578,A -85,B 0,C 180,E1 -14319.717,E2 -14319.717} C_VEL
LIN {X 0,Y 340.84,Z 336.655,A -85,B 0,C 180,E1 -14320.846,E2 -14320.846} C_VEL
LIN {X 0,Y 340.83,Z 336.652,A -85,B 0,C 180,E1 -14322.267,E2 -14322.267} C_VEL
LIN {X 0,Y 340.144,Z 336.743,A -85,B 0,C 180,E1 -14323.253,E2 -14323.253} C_VEL
LIN {X 0,Y 337.266,Z 337.103,A -85,B 0,C 180,E1 -14324.857,E2 -14324.857} C_VEL
LIN {X 0,Y 334.836,Z 337.407,A -85,B 0,C 180,E1 -14326.156,E2 -14326.156} C_VEL
LIN {X 0,Y 333.793,Z 337.535,A -85,B 0,C 180,E1 -14327.161,E2 -14327.161} C_VEL
LIN {X 0,Y 333.708,Z 337.542,A -85,B 0,C 180,E1 -14327.502,E2 -14327.502} C_VEL
LIN {X 0,Y 333.666,Z 337.55,A -85,B 0,C 180,E1 -14330.983,E2 -14330.983} C_VEL
LIN {X 0,Y 333.686,Z 337.547,A -85,B 0,C 180,E1 -14335.09,E2 -14335.09} C_VEL
LIN {X 0,Y 333.649,Z 337.552,A -85,B 0,C 180,E1 -14338.979,E2 -14338.979} C_VEL
LIN {X 0,Y 333.639,Z 337.55,A -85,B 0,C 180,E1 -14342.587,E2 -14342.587} C_VEL
LIN {X 0,Y 333.672,Z 337.542,A -85,B 0,C 180,E1 -14346.14,E2 -14346.14} C_VEL
LIN {X 0,Y 333.619,Z 337.552,A -85,B 0,C 180,E1 -14349.197,E2 -14349.197} C_VEL
LIN {X 0,Y 333.626,Z 337.552,A -85,B 0,C 180,E1 -14352.5,E2 -14352.5} C_VEL
LIN {X 0,Y 333.593,Z 337.551,A -85,B 0,C 180,E1 -14355.955,E2 -14355.955} C_VEL
LIN {X 0,Y 333.602,Z 337.552,A -85,B 0,C 180,E1 -14359.326,E2 -14359.326} C_VEL
LIN {X 0,Y 333.663,Z 337.541,A -85,B 0,C 180,E1 -14363.17,E2 -14363.17} C_VEL
LIN {X 0,Y 333.675,Z 337.54,A -85,B 0,C 180,E1 -14365.342,E2 -14365.342} C_VEL
LIN {X 0,Y 333.631,Z 337.551,A -85,B 0,C 180,E1 -14368.223,E2 -14368.223} C_VEL
LIN {X 0,Y 333.633,Z 337.549,A -85,B 0,C 180,E1 -14371.021,E2 -14371.021} C_VEL
LIN {X 0,Y 333.657,Z 337.547,A -85,B 0,C 180,E1 -14374.924,E2 -14374.924} C_VEL
LIN {X 0,Y 333.656,Z 337.545,A -85,B 0,C 180,E1 -14379.018,E2 -14379.018} C_VEL
LIN {X 0,Y 333.727,Z 337.537,A -85,B 0,C 180,E1 -14381.586,E2 -14381.586} C_VEL
LIN {X 0,Y 333.776,Z 337.528,A -85,B 0,C 180,E1 -14385.601,E2 -14385.601} C_VEL
LIN {X 0,Y 333.82,Z 337.521,A -85,B 0,C 180,E1 -14389.078,E2 -14389.078} C_VEL
LIN {X 0,Y 333.961,Z 337.508,A -85,B 0,C 180,E1 -14392.747,E2 -14392.747} C_VEL
LIN {X 0,Y 333.796,Z 337.527,A -85,B 0,C 180,E1 -14395.169,E2 -14395.169} C_VEL
LIN {X 0,Y 334.098,Z 337.49,A -85,B 0,C 180,E1 -14397.589,E2 -14397.589} C_VEL
LIN {X 0,Y 334.19,Z 337.478,A -85,B 0,C 180,E1 -14400,E2 -14400} C_VEL
LIN {X 0,Y 334.076,Z 337.493,A -85,B 0,C 180,E1 -14402.412,E2 -14402.412} C_VEL
LIN {X 0,Y 334.004,Z 337.506,A -85,B 0,C 180,E1 -14406.04,E2 -14406.04} C_VEL
LIN {X 0,Y 333.825,Z 337.528,A -85,B 0,C 180,E1 -14409.697,E2 -14409.697} C_VEL
LIN {X 0,Y 333.801,Z 337.529,A -85,B 0,C 180,E1 -14413.392,E2 -14413.392} C_VEL
LIN {X 0,Y 333.751,Z 337.535,A -85,B 0,C 180,E1 -14417.146,E2 -14417.146} C_VEL
LIN {X 0,Y 333.741,Z 337.539,A -85,B 0,C 180,E1 -14419.69,E2 -14419.69} C_VEL
LIN {X 0,Y 333.697,Z 337.541,A -85,B 0,C 180,E1 -14422.278,E2 -14422.278} C_VEL
LIN {X 0,Y 333.74,Z 337.535,A -85,B 0,C 180,E1 -14426.246,E2 -14426.246} C_VEL
LIN {X 0,Y 333.695,Z 337.541,A -85,B 0,C 180,E1 -14428.974,E2 -14428.974} C_VEL
LIN {X 0,Y 333.648,Z 337.546,A -85,B 0,C 180,E1 -14432.587,E2 -14432.587} C_VEL
LIN {X 0,Y 333.681,Z 337.542,A -85,B 0,C 180,E1 -14436.139,E2 -14436.139} C_VEL
LIN {X 0,Y 333.652,Z 337.548,A -85,B 0,C 180,E1 -14439.192,E2 -14439.192} C_VEL
LIN {X 0,Y 333.637,Z 337.548,A -85,B 0,C 180,E1 -14442.5,E2 -14442.5} C_VEL
LIN {X 0,Y 333.627,Z 337.549,A -85,B 0,C 180,E1 -14445.959,E2 -14445.959} C_VEL
LIN {X 0,Y 333.652,Z 337.55,A -85,B 0,C 180,E1 -14449.315,E2 -14449.315} C_VEL
LIN {X 0,Y 333.669,Z 337.55,A -85,B 0,C 180,E1 -14453.167,E2 -14453.167} C_VEL
LIN {X 0,Y 333.726,Z 337.7,A -85,B 0,C 180,E1 -14455.712,E2 -14455.712} C_VEL
LIN {X 0,Y 336.983,Z 351.937,A -85,B 0,C 180,E1 -14459.355,E2 -14459.355} C_VEL
LIN {X 0,Y 339.372,Z 363.611,A -85,B 0,C 180,E1 -14462.162,E2 -14462.162} C_VEL
LIN {X 0,Y 343.655,Z 388.39,A -85,B 0,C 180,E1 -14463.033,E2 -14463.033} C_VEL
LIN {X 0,Y 346.521,Z 407.156,A -85,B 0,C 180,E1 -14463.65,E2 -14463.65} C_VEL
LIN {X 0,Y 344.338,Z 501.042,A -85,B 0,C 180,E1 -14465.626,E2 -14465.626} C_VEL
LIN {X 0,Y 343.583,Z 515.234,A -85,B 0,C 180,E1 -14466.131,E2 -14466.131} C_VEL
LIN {X 0,Y 342.36,Z 529.553,A -85,B 0,C 180,E1 -14466.883,E2 -14466.883} C_VEL
LIN {X 0,Y 341.195,Z 541.935,A -85,B 0,C 180,E1 -14467.759,E2 -14467.759} C_VEL
LIN {X 0,Y 339.769,Z 555.068,A -85,B 0,C 180,E1 -14468.952,E2 -14468.952} C_VEL
LIN {X 0,Y 338.254,Z 566.704,A -85,B 0,C 180,E1 -14470.266,E2 -14470.266} C_VEL
LIN {X 0,Y 336.813,Z 577.495,A -85,B 0,C 180,E1 -14471.759,E2 -14471.759} C_VEL
LIN {X 0,Y 335.399,Z 588.188,A -85,B 0,C 180,E1 -14473.567,E2 -14473.567} C_VEL
LIN {X 0,Y 334.282,Z 596.999,A -85,B 0,C 180,E1 -14475.386,E2 -14475.386} C_VEL
LIN {X 0,Y 333.479,Z 604.312,A -85,B 0,C 180,E1 -14477.214,E2 -14477.214} C_VEL
LIN {X 0,Y 332.741,Z 610.369,A -85,B 0,C 180,E1 -14479.041,E2 -14479.041} C_VEL
LIN {X 0,Y 332.357,Z 615.372,A -85,B 0,C 180,E1 -14480.874,E2 -14480.874} C_VEL
LIN {X 0,Y 332.099,Z 620.514,A -85,B 0,C 180,E1 -14483.315,E2 -14483.315} C_VEL
LIN {X 0,Y 331.994,Z 623.378,A -85,B 0,C 180,E1 -14485.142,E2 -14485.142} C_VEL
LIN {X 0,Y 331.968,Z 625.878,A -85,B 0,C 180,E1 -14487.572,E2 -14487.572} C_VEL
LIN {X 0,Y 332.045,Z 627.002,A -85,B 0,C 180,E1 -14489.999,E2 -14489.999} C_VEL
LIN {X 0,Y 331.938,Z 626.77,A -85,B 0,C 180,E1 -14492.426,E2 -14492.426} C_VEL
LIN {X 0,Y 331.985,Z 626.155,A -85,B 0,C 180,E1 -14493.64,E2 -14493.64} C_VEL
LIN {X 0,Y 332.043,Z 623.913,A -85,B 0,C 180,E1 -14496.074,E2 -14496.074} C_VEL
LIN {X 0,Y 332.321,Z 620.28,A -85,B 0,C 180,E1 -14498.512,E2 -14498.512} C_VEL
LIN {X 0,Y 332.875,Z 615.162,A -85,B 0,C 180,E1 -14500.953,E2 -14500.953} C_VEL
LIN {X 0,Y 334.06,Z 608.416,A -85,B 0,C 180,E1 -14503.379,E2 -14503.379} C_VEL
LIN {X 0,Y 335.156,Z 601.426,A -85,B 0,C 180,E1 -14505.376,E2 -14505.376} C_VEL
LIN {X 0,Y 336.676,Z 593.155,A -85,B 0,C 180,E1 -14507.304,E2 -14507.304} C_VEL
LIN {X 0,Y 338.469,Z 583.829,A -85,B 0,C 180,E1 -14509.088,E2 -14509.088} C_VEL
LIN {X 0,Y 340.642,Z 572.483,A -85,B 0,C 180,E1 -14510.847,E2 -14510.847} C_VEL
LIN {X 0,Y 342.63,Z 561.44,A -85,B 0,C 180,E1 -14512.243,E2 -14512.243} C_VEL
LIN {X 0,Y 344.407,Z 549.862,A -85,B 0,C 180,E1 -14513.446,E2 -14513.446} C_VEL
LIN {X 0,Y 346.035,Z 537.909,A -85,B 0,C 180,E1 -14514.444,E2 -14514.444} C_VEL
LIN {X 0,Y 347.657,Z 524.841,A -85,B 0,C 180,E1 -14515.279,E2 -14515.279} C_VEL
LIN {X 0,Y 348.962,Z 510.797,A -85,B 0,C 180,E1 -14515.937,E2 -14515.937} C_VEL
LIN {X 0,Y 349.87,Z 496.044,A -85,B 0,C 180,E1 -14516.386,E2 -14516.386} C_VEL
LIN {X 0,Y 352.437,Z 408.427,A -85,B 0,C 180,E1 -14518.237,E2 -14518.237} C_VEL
LIN {X 0,Y 349.063,Z 388.404,A -85,B 0,C 180,E1 -14519.079,E2 -14519.079} C_VEL
LIN {X 0,Y 346.212,Z 375.633,A -85,B 0,C 180,E1 -14519.708,E2 -14519.708} C_VEL
LIN {X 0,Y 340.094,Z 362.242,A -85,B 0,C 180,E1 -14520.77,E2 -14520.77} C_VEL
LIN {X 0,Y 337.476,Z 351.102,A -85,B 0,C 180,E1 -14523.943,E2 -14523.943} C_VEL
LIN {X 0,Y 334.637,Z 341.067,A -85,B 0,C 180,E1 -14527.053,E2 -14527.053} C_VEL
LIN {X 0,Y 333.694,Z 337.537,A -85,B 0,C 180,E1 -14528.218,E2 -14528.218} C_VEL
LIN {X 0,Y 333.67,Z 337.536,A -85,B 0,C 180,E1 -14532.375,E2 -14532.375} C_VEL
LIN {X 0,Y 333.593,Z 337.541,A -85,B 0,C 180,E1 -14535.954,E2 -14535.954} C_VEL
LIN {X 0,Y 333.643,Z 337.539,A -85,B 0,C 180,E1 -14539.314,E2 -14539.314} C_VEL
LIN {X 0,Y 333.661,Z 337.547,A -85,B 0,C 180,E1 -14543.166,E2 -14543.166} C_VEL
LIN {X 0,Y 333.633,Z 337.546,A -85,B 0,C 180,E1 -14546.791,E2 -14546.791} C_VEL
LIN {X 0,Y 333.697,Z 337.54,A -85,B 0,C 180,E1 -14549.709,E2 -14549.709} C_VEL
LIN {X 0,Y 333.738,Z 337.537,A -85,B 0,C 180,E1 -14552.4,E2 -14552.4} C_VEL
LIN {X 0,Y 333.719,Z 337.54,A -85,B 0,C 180,E1 -14555.09,E2 -14555.09} C_VEL
LIN {X 0,Y 333.673,Z 337.546,A -85,B 0,C 180,E1 -14559.018,E2 -14559.018} C_VEL
LIN {X 0,Y 333.786,Z 337.524,A -85,B 0,C 180,E1 -14561.589,E2 -14561.589} C_VEL
LIN {X 0,Y 333.801,Z 337.522,A -85,B 0,C 180,E1 -14565.576,E2 -14565.576} C_VEL
LIN {X 0,Y 333.825,Z 337.516,A -85,B 0,C 180,E1 -14569.077,E2 -14569.077} C_VEL
LIN {X 0,Y 334.016,Z 337.494,A -85,B 0,C 180,E1 -14572.747,E2 -14572.747} C_VEL
LIN {X 0,Y 333.786,Z 337.532,A -85,B 0,C 180,E1 -14575.168,E2 -14575.168} C_VEL
LIN {X 0,Y 334.061,Z 337.49,A -85,B 0,C 180,E1 -14577.588,E2 -14577.588} C_VEL
LIN {X 0,Y 334.05,Z 337.491,A -85,B 0,C 180,E1 -14581.205,E2 -14581.205} C_VEL
LIN {X 0,Y 334.063,Z 337.496,A -85,B 0,C 180,E1 -14582.411,E2 -14582.411} C_VEL
LIN {X 0,Y 333.946,Z 337.508,A -85,B 0,C 180,E1 -14586.482,E2 -14586.482} C_VEL
LIN {X 0,Y 333.81,Z 337.524,A -85,B 0,C 180,E1 -14589.696,E2 -14589.696} C_VEL
LIN {X 0,Y 333.783,Z 337.528,A -85,B 0,C 180,E1 -14593.392,E2 -14593.392} C_VEL
LIN {X 0,Y 333.708,Z 337.539,A -85,B 0,C 180,E1 -14597.148,E2 -14597.148} C_VEL
LIN {X 0,Y 333.662,Z 337.544,A -85,B 0,C 180,E1 -14599.694,E2 -14599.694} C_VEL
LIN {X 0,Y 333.651,Z 337.551,A -85,B 0,C 180,E1 -14603.591,E2 -14603.591} C_VEL
LIN {X 0,Y 333.647,Z 337.551,A -85,B 0,C 180,E1 -14606.253,E2 -14606.253} C_VEL
LIN {X 0,Y 333.653,Z 337.551,A -85,B 0,C 180,E1 -14610.278,E2 -14610.278} C_VEL
LIN {X 0,Y 333.628,Z 337.544,A -85,B 0,C 180,E1 -14613.209,E2 -14613.209} C_VEL
LIN {X 0,Y 333.667,Z 337.542,A -85,B 0,C 180,E1 -14616.139,E2 -14616.139} C_VEL
LIN {X 0,Y 333.696,Z 337.733,A -85,B 0,C 180,E1 -14619.062,E2 -14619.062} C_VEL
LIN {X 0,Y 334.912,Z 342.277,A -85,B 0,C 180,E1 -14620.649,E2 -14620.649} C_VEL
LIN {X 0,Y 343.869,Z 358.872,A -85,B 0,C 180,E1 -14622.17,E2 -14622.17} C_VEL
LIN {X 0,Y 351.196,Z 374.162,A -85,B 0,C 180,E1 -14623.369,E2 -14623.369} C_VEL
LIN {X 0,Y 353.253,Z 379.322,A -85,B 0,C 180,E1 -14623.712,E2 -14623.712} C_VEL
LIN {X 0,Y 350.245,Z 477.549,A -85,B 0,C 180,E1 -14625.798,E2 -14625.798} C_VEL
LIN {X 0,Y 349.408,Z 491.429,A -85,B 0,C 180,E1 -14626.296,E2 -14626.296} C_VEL
LIN {X 0,Y 348.264,Z 504.475,A -85,B 0,C 180,E1 -14626.975,E2 -14626.975} C_VEL
LIN {X 0,Y 346.92,Z 517.055,A -85,B 0,C 180,E1 -14627.853,E2 -14627.853} C_VEL
LIN {X 0,Y 345.124,Z 530.021,A -85,B 0,C 180,E1 -14629.009,E2 -14629.009} C_VEL
LIN {X 0,Y 343.133,Z 542.363,A -85,B 0,C 180,E1 -14630.396,E2 -14630.396} C_VEL
LIN {X 0,Y 341.122,Z 553.904,A -85,B 0,C 180,E1 -14632.013,E2 -14632.013} C_VEL
LIN {X 0,Y 339.36,Z 563.288,A -85,B 0,C 180,E1 -14633.621,E2 -14633.621} C_VEL
LIN {X 0,Y 337.617,Z 572.092,A -85,B 0,C 180,E1 -14635.443,E2 -14635.443} C_VEL
LIN {X 0,Y 336.039,Z 579.896,A -85,B 0,C 180,E1 -14637.417,E2 -14637.417} C_VEL
LIN {X 0,Y 334.603,Z 587.206,A -85,B 0,C 180,E1 -14639.73,E2 -14639.73} C_VEL
LIN {X 0,Y 333.682,Z 592.11,A -85,B 0,C 180,E1 -14641.715,E2 -14641.715} C_VEL
LIN {X 0,Y 332.95,Z 595.926,A -85,B 0,C 180,E1 -14643.689,E2 -14643.689} C_VEL
LIN {X 0,Y 332.514,Z 598.415,A -85,B 0,C 180,E1 -14645.345,E2 -14645.345} C_VEL
LIN {X 0,Y 332.086,Z 600.736,A -85,B 0,C 180,E1 -14647.61,E2 -14647.61} C_VEL
LIN {X 0,Y 331.979,Z 601.533,A -85,B 0,C 180,E1 -14648.908,E2 -14648.908} C_VEL
LIN {X 0,Y 331.815,Z 602.013,A -85,B 0,C 180,E1 -14651.477,E2 -14651.477} C_VEL
LIN {X 0,Y 331.838,Z 601.71,A -85,B 0,C 180,E1 -14652.753,E2 -14652.753} C_VEL
LIN {X 0,Y 331.868,Z 600.048,A -85,B 0,C 180,E1 -14655.28,E2 -14655.28} C_VEL
LIN {X 0,Y 332.058,Z 598.361,A -85,B 0,C 180,E1 -14656.8,E2 -14656.8} C_VEL
LIN {X 0,Y 332.418,Z 594.844,A -85,B 0,C 180,E1 -14659.032,E2 -14659.032} C_VEL
LIN {X 0,Y 332.814,Z 590.922,A -85,B 0,C 180,E1 -14660.888,E2 -14660.888} C_VEL
LIN {X 0,Y 333.436,Z 586.065,A -85,B 0,C 180,E1 -14662.736,E2 -14662.736} C_VEL
LIN {X 0,Y 334.227,Z 579.073,A -85,B 0,C 180,E1 -14664.874,E2 -14664.874} C_VEL
LIN {X 0,Y 335.433,Z 570.385,A -85,B 0,C 180,E1 -14666.999,E2 -14666.999} C_VEL
LIN {X 0,Y 336.71,Z 561.306,A -85,B 0,C 180,E1 -14668.805,E2 -14668.805} C_VEL
LIN {X 0,Y 337.856,Z 552.304,A -85,B 0,C 180,E1 -14670.299,E2 -14670.299} C_VEL
LIN {X 0,Y 339.298,Z 541.526,A -85,B 0,C 180,E1 -14671.782,E2 -14671.782} C_VEL
LIN {X 0,Y 340.669,Z 529.778,A -85,B 0,C 180,E1 -14673.105,E2 -14673.105} C_VEL
LIN {X 0,Y 342.029,Z 516.826,A -85,B 0,C 180,E1 -14674.273,E2 -14674.273} C_VEL
LIN {X 0,Y 343.17,Z 503.342,A -85,B 0,C 180,E1 -14675.215,E2 -14675.215} C_VEL
LIN {X 0,Y 344.041,Z 489.241,A -85,B 0,C 180,E1 -14675.937,E2 -14675.937} C_VEL
LIN {X 0,Y 344.716,Z 475.547,A -85,B 0,C 180,E1 -14676.403,E2 -14676.403} C_VEL
LIN {X 0,Y 347.097,Z 373.591,A -85,B 0,C 180,E1 -14678.543,E2 -14678.543} C_VEL
LIN {X 0,Y 338.15,Z 349.731,A -85,B 0,C 180,E1 -14679.732,E2 -14679.732} C_VEL
LIN {X 0,Y 334.569,Z 340.913,A -85,B 0,C 180,E1 -14680.234,E2 -14680.234} C_VEL
LIN {X 0,Y 333.799,Z 337.529,A -85,B 0,C 180,E1 -14681.231,E2 -14681.231} C_VEL
LIN {X 0,Y 333.807,Z 337.528,A -85,B 0,C 180,E1 -14684.635,E2 -14684.635} C_VEL
LIN {X 0,Y 333.708,Z 337.542,A -85,B 0,C 180,E1 -14687.502,E2 -14687.502} C_VEL
LIN {X 0,Y 333.039,Z 337.626,A -85,B 0,C 180,E1 -14688.508,E2 -14688.508} C_VEL
LIN {X 0,Y 330.178,Z 337.985,A -85,B 0,C 180,E1 -14690.145,E2 -14690.145} C_VEL
LIN {X 0,Y 327.743,Z 338.292,A -85,B 0,C 180,E1 -14691.471,E2 -14691.471} C_VEL
LIN {X 0,Y 326.685,Z 338.42,A -85,B 0,C 180,E1 -14692.498,E2 -14692.498} C_VEL
LIN {X 0,Y 326.592,Z 338.429,A -85,B 0,C 180,E1 -14692.846,E2 -14692.846} C_VEL
LIN {X 0,Y 326.632,Z 338.423,A -85,B 0,C 180,E1 -14695.49,E2 -14695.49} C_VEL
LIN {X 0,Y 326.587,Z 338.427,A -85,B 0,C 180,E1 -14699.667,E2 -14699.667} C_VEL
LIN {X 0,Y 326.614,Z 338.428,A -85,B 0,C 180,E1 -14702.946,E2 -14702.946} C_VEL
LIN {X 0,Y 326.61,Z 338.422,A -85,B 0,C 180,E1 -14705.521,E2 -14705.521} C_VEL
LIN {X 0,Y 326.587,Z 338.428,A -85,B 0,C 180,E1 -14709.223,E2 -14709.223} C_VEL
LIN {X 0,Y 326.571,Z 338.428,A -85,B 0,C 180,E1 -14712.972,E2 -14712.972} C_VEL
LIN {X 0,Y 326.572,Z 338.43,A -85,B 0,C 180,E1 -14717.03,E2 -14717.03} C_VEL
LIN {X 0,Y 326.586,Z 338.428,A -85,B 0,C 180,E1 -14720.779,E2 -14720.779} C_VEL
LIN {X 0,Y 326.612,Z 338.42,A -85,B 0,C 180,E1 -14724.481,E2 -14724.481} C_VEL
LIN {X 0,Y 326.609,Z 338.422,A -85,B 0,C 180,E1 -14727.456,E2 -14727.456} C_VEL
LIN {X 0,Y 326.583,Z 338.431,A -85,B 0,C 180,E1 -14730.334,E2 -14730.334} C_VEL
LIN {X 0,Y 326.598,Z 338.424,A -85,B 0,C 180,E1 -14733.135,E2 -14733.135} C_VEL
LIN {X 0,Y 326.592,Z 338.424,A -85,B 0,C 180,E1 -14737.211,E2 -14737.211} C_VEL
LIN {X 0,Y 326.673,Z 338.415,A -85,B 0,C 180,E1 -14741.195,E2 -14741.195} C_VEL
LIN {X 0,Y 326.728,Z 338.405,A -85,B 0,C 180,E1 -14745.46,E2 -14745.46} C_VEL
LIN {X 0,Y 326.761,Z 338.4,A -85,B 0,C 180,E1 -14748.839,E2 -14748.839} C_VEL
LIN {X 0,Y 326.917,Z 338.386,A -85,B 0,C 180,E1 -14752.589,E2 -14752.589} C_VEL
LIN {X 0,Y 326.763,Z 338.403,A -85,B 0,C 180,E1 -14755.065,E2 -14755.065} C_VEL
LIN {X 0,Y 327.038,Z 338.368,A -85,B 0,C 180,E1 -14757.537,E2 -14757.537} C_VEL
LIN {X 0,Y 327.143,Z 338.354,A -85,B 0,C 180,E1 -14760,E2 -14760} C_VEL
LIN {X 0,Y 327.019,Z 338.372,A -85,B 0,C 180,E1 -14762.464,E2 -14762.464} C_VEL
LIN {X 0,Y 326.957,Z 338.382,A -85,B 0,C 180,E1 -14766.17,E2 -14766.17} C_VEL
LIN {X 0,Y 326.788,Z 338.406,A -85,B 0,C 180,E1 -14769.907,E2 -14769.907} C_VEL
LIN {X 0,Y 326.764,Z 338.408,A -85,B 0,C 180,E1 -14773.686,E2 -14773.686} C_VEL
LIN {X 0,Y 326.704,Z 338.415,A -85,B 0,C 180,E1 -14777.528,E2 -14777.528} C_VEL
LIN {X 0,Y 326.667,Z 338.416,A -85,B 0,C 180,E1 -14780.135,E2 -14780.135} C_VEL
LIN {X 0,Y 326.657,Z 338.417,A -85,B 0,C 180,E1 -14784.129,E2 -14784.129} C_VEL
LIN {X 0,Y 326.687,Z 338.413,A -85,B 0,C 180,E1 -14786.858,E2 -14786.858} C_VEL
LIN {X 0,Y 326.639,Z 338.419,A -85,B 0,C 180,E1 -14790.61,E2 -14790.61} C_VEL
LIN {X 0,Y 326.611,Z 338.424,A -85,B 0,C 180,E1 -14794.019,E2 -14794.019} C_VEL
LIN {X 0,Y 326.633,Z 338.424,A -85,B 0,C 180,E1 -14797.239,E2 -14797.239} C_VEL
LIN {X 0,Y 326.583,Z 338.431,A -85,B 0,C 180,E1 -14801.131,E2 -14801.131} C_VEL
LIN {X 0,Y 326.56,Z 338.431,A -85,B 0,C 180,E1 -14804.748,E2 -14804.748} C_VEL
LIN {X 0,Y 326.581,Z 338.428,A -85,B 0,C 180,E1 -14808.154,E2 -14808.154} C_VEL
LIN {X 0,Y 326.628,Z 338.426,A -85,B 0,C 180,E1 -14811.391,E2 -14811.391} C_VEL
LIN {X 0,Y 326.669,Z 338.559,A -85,B 0,C 180,E1 -14815.287,E2 -14815.287} C_VEL
LIN {X 0,Y 329.722,Z 351.915,A -85,B 0,C 180,E1 -14818.788,E2 -14818.788} C_VEL
LIN {X 0,Y 332.174,Z 363.296,A -85,B 0,C 180,E1 -14821.613,E2 -14821.613} C_VEL
LIN {X 0,Y 333.782,Z 368.833,A -85,B 0,C 180,E1 -14821.866,E2 -14821.866} C_VEL
LIN {X 0,Y 339.928,Z 407.171,A -85,B 0,C 180,E1 -14823.199,E2 -14823.199} C_VEL
LIN {X 0,Y 337.708,Z 500.414,A -85,B 0,C 180,E1 -14825.198,E2 -14825.198} C_VEL
LIN {X 0,Y 336.945,Z 514.781,A -85,B 0,C 180,E1 -14825.713,E2 -14825.713} C_VEL
LIN {X 0,Y 335.7,Z 529.153,A -85,B 0,C 180,E1 -14826.478,E2 -14826.478} C_VEL
LIN {X 0,Y 334.373,Z 542.444,A -85,B 0,C 180,E1 -14827.443,E2 -14827.443} C_VEL
LIN {X 0,Y 332.868,Z 555.74,A -85,B 0,C 180,E1 -14828.691,E2 -14828.691} C_VEL
LIN {X 0,Y 331.348,Z 566.959,A -85,B 0,C 180,E1 -14829.999,E2 -14829.999} C_VEL
LIN {X 0,Y 329.978,Z 576.67,A -85,B 0,C 180,E1 -14831.368,E2 -14831.368} C_VEL
LIN {X 0,Y 328.503,Z 587.456,A -85,B 0,C 180,E1 -14833.212,E2 -14833.212} C_VEL
LIN {X 0,Y 327.206,Z 597.375,A -85,B 0,C 180,E1 -14835.302,E2 -14835.302} C_VEL
LIN {X 0,Y 326.374,Z 604.863,A -85,B 0,C 180,E1 -14837.248,E2 -14837.248} C_VEL
LIN {X 0,Y 325.543,Z 611.674,A -85,B 0,C 180,E1 -14839.425,E2 -14839.425} C_VEL
LIN {X 0,Y 325.124,Z 617.705,A -85,B 0,C 180,E1 -14841.922,E2 -14841.922} C_VEL
LIN {X 0,Y 324.951,Z 621.803,A -85,B 0,C 180,E1 -14844.204,E2 -14844.204} C_VEL
LIN {X 0,Y 324.93,Z 624.46,A -85,B 0,C 180,E1 -14846.279,E2 -14846.279} C_VEL
LIN {X 0,Y 324.916,Z 626.308,A -85,B 0,C 180,E1 -14848.759,E2 -14848.759} C_VEL
LIN {X 0,Y 324.95,Z 626.722,A -85,B 0,C 180,E1 -14849.999,E2 -14849.999} C_VEL
LIN {X 0,Y 324.856,Z 626.533,A -85,B 0,C 180,E1 -14852.479,E2 -14852.479} C_VEL
LIN {X 0,Y 324.874,Z 625.008,A -85,B 0,C 180,E1 -14854.963,E2 -14854.963} C_VEL
LIN {X 0,Y 325.079,Z 622.125,A -85,B 0,C 180,E1 -14857.452,E2 -14857.452} C_VEL
LIN {X 0,Y 325.511,Z 617.81,A -85,B 0,C 180,E1 -14859.945,E2 -14859.945} C_VEL
LIN {X 0,Y 326.441,Z 611.952,A -85,B 0,C 180,E1 -14862.431,E2 -14862.431} C_VEL
LIN {X 0,Y 327.579,Z 605.389,A -85,B 0,C 180,E1 -14864.6,E2 -14864.6} C_VEL
LIN {X 0,Y 329.059,Z 597.299,A -85,B 0,C 180,E1 -14866.757,E2 -14866.757} C_VEL
LIN {X 0,Y 330.758,Z 588.865,A -85,B 0,C 180,E1 -14868.584,E2 -14868.584} C_VEL
LIN {X 0,Y 332.873,Z 578.738,A -85,B 0,C 180,E1 -14870.386,E2 -14870.386} C_VEL
LIN {X 0,Y 335.031,Z 567.442,A -85,B 0,C 180,E1 -14872.021,E2 -14872.021} C_VEL
LIN {X 0,Y 336.992,Z 556.263,A -85,B 0,C 180,E1 -14873.342,E2 -14873.342} C_VEL
LIN {X 0,Y 338.908,Z 544.107,A -85,B 0,C 180,E1 -14874.502,E2 -14874.502} C_VEL
LIN {X 0,Y 340.592,Z 531.762,A -85,B 0,C 180,E1 -14875.432,E2 -14875.432} C_VEL
LIN {X 0,Y 342.155,Z 518.085,A -85,B 0,C 180,E1 -14876.206,E2 -14876.206} C_VEL
LIN {X 0,Y 343.372,Z 503.96,A -85,B 0,C 180,E1 -14876.761,E2 -14876.761} C_VEL
LIN {X 0,Y 344.141,Z 484.74,A -85,B 0,C 180,E1 -14877.229,E2 -14877.229} C_VEL
LIN {X 0,Y 346.362,Z 408.715,A -85,B 0,C 180,E1 -14878.867,E2 -14878.867} C_VEL
LIN {X 0,Y 343.055,Z 389.519,A -85,B 0,C 180,E1 -14879.713,E2 -14879.713} C_VEL
LIN {X 0,Y 340.555,Z 378.318,A -85,B 0,C 180,E1 -14880.285,E2 -14880.285} C_VEL
LIN {X 0,Y 334.613,Z 365.685,A -85,B 0,C 180,E1 -14881.331,E2 -14881.331} C_VEL
LIN {X 0,Y 332.894,Z 361.918,A -85,B 0,C 180,E1 -14881.658,E2 -14881.658} C_VEL
LIN {X 0,Y 330.335,Z 351.482,A -85,B 0,C 180,E1 -14884.754,E2 -14884.754} C_VEL
LIN {X 0,Y 327.361,Z 340.989,A -85,B 0,C 180,E1 -14888.143,E2 -14888.143} C_VEL
LIN {X 0,Y 326.627,Z 338.416,A -85,B 0,C 180,E1 -14889.024,E2 -14889.024} C_VEL
LIN {X 0,Y 326.596,Z 338.422,A -85,B 0,C 180,E1 -14892.975,E2 -14892.975} C_VEL
LIN {X 0,Y 326.572,Z 338.423,A -85,B 0,C 180,E1 -14897.027,E2 -14897.027} C_VEL
LIN {X 0,Y 326.607,Z 338.408,A -85,B 0,C 180,E1 -14900.771,E2 -14900.771} C_VEL
LIN {X 0,Y 326.607,Z 338.423,A -85,B 0,C 180,E1 -14904.479,E2 -14904.479} C_VEL
LIN {X 0,Y 326.604,Z 338.421,A -85,B 0,C 180,E1 -14907.455,E2 -14907.455} C_VEL
LIN {X 0,Y 326.655,Z 338.415,A -85,B 0,C 180,E1 -14910.34,E2 -14910.34} C_VEL
LIN {X 0,Y 326.683,Z 338.414,A -85,B 0,C 180,E1 -14914.515,E2 -14914.515} C_VEL
LIN {X 0,Y 326.639,Z 338.423,A -85,B 0,C 180,E1 -14918.544,E2 -14918.544} C_VEL
LIN {X 0,Y 326.737,Z 338.4,A -85,B 0,C 180,E1 -14921.177,E2 -14921.177} C_VEL
LIN {X 0,Y 326.756,Z 338.399,A -85,B 0,C 180,E1 -14925.432,E2 -14925.432} C_VEL
LIN {X 0,Y 326.761,Z 338.396,A -85,B 0,C 180,E1 -14928.838,E2 -14928.838} C_VEL
LIN {X 0,Y 326.97,Z 338.372,A -85,B 0,C 180,E1 -14932.59,E2 -14932.59} C_VEL
LIN {X 0,Y 326.755,Z 338.407,A -85,B 0,C 180,E1 -14935.064,E2 -14935.064} C_VEL
LIN {X 0,Y 327.005,Z 338.368,A -85,B 0,C 180,E1 -14937.536,E2 -14937.536} C_VEL
LIN {X 0,Y 327.02,Z 338.367,A -85,B 0,C 180,E1 -14941.231,E2 -14941.231} C_VEL
LIN {X 0,Y 326.754,Z 338.408,A -85,B 0,C 180,E1 -14943.699,E2 -14943.699} C_VEL
LIN {X 0,Y 326.909,Z 338.385,A -85,B 0,C 180,E1 -14946.47,E2 -14946.47} C_VEL
LIN {X 0,Y 326.773,Z 338.402,A -85,B 0,C 180,E1 -14949.907,E2 -14949.907} C_VEL
LIN {X 0,Y 326.747,Z 338.407,A -85,B 0,C 180,E1 -14953.685,E2 -14953.685} C_VEL
LIN {X 0,Y 326.654,Z 338.423,A -85,B 0,C 180,E1 -14957.53,E2 -14957.53} C_VEL
LIN {X 0,Y 326.609,Z 338.424,A -85,B 0,C 180,E1 -14961.457,E2 -14961.457} C_VEL
LIN {X 0,Y 326.625,Z 338.423,A -85,B 0,C 180,E1 -14965.489,E2 -14965.489} C_VEL
LIN {X 0,Y 326.608,Z 338.417,A -85,B 0,C 180,E1 -14969.664,E2 -14969.664} C_VEL
LIN {X 0,Y 326.608,Z 338.417,A -85,B 0,C 180,E1 -14972.946,E2 -14972.946} C_VEL
LIN {X 0,Y 326.604,Z 338.428,A -85,B 0,C 180,E1 -14975.52,E2 -14975.52} C_VEL
LIN {X 0,Y 326.606,Z 338.53,A -85,B 0,C 180,E1 -14978.237,E2 -14978.237} C_VEL
LIN {X 0,Y 327.85,Z 342.778,A -85,B 0,C 180,E1 -14979.742,E2 -14979.742} C_VEL
LIN {X 0,Y 337.319,Z 359.99,A -85,B 0,C 180,E1 -14981.421,E2 -14981.421} C_VEL
LIN {X 0,Y 344.791,Z 375.257,A -85,B 0,C 180,E1 -14982.689,E2 -14982.689} C_VEL
LIN {X 0,Y 347.179,Z 380.887,A -85,B 0,C 180,E1 -14983.097,E2 -14983.097} C_VEL
LIN {X 0,Y 344.539,Z 465.699,A -85,B 0,C 180,E1 -14984.914,E2 -14984.914} C_VEL
LIN {X 0,Y 343.864,Z 482.448,A -85,B 0,C 180,E1 -14985.344,E2 -14985.344} C_VEL
LIN {X 0,Y 342.839,Z 496.617,A -85,B 0,C 180,E1 -14985.938,E2 -14985.938} C_VEL
LIN {X 0,Y 341.532,Z 509.868,A -85,B 0,C 180,E1 -14986.727,E2 -14986.727} C_VEL
LIN {X 0,Y 339.906,Z 523.077,A -85,B 0,C 180,E1 -14987.768,E2 -14987.768} C_VEL
LIN {X 0,Y 337.921,Z 536,A -85,B 0,C 180,E1 -14989.072,E2 -14989.072} C_VEL
LIN {X 0,Y 335.899,Z 547.389,A -85,B 0,C 180,E1 -14990.502,E2 -14990.502} C_VEL
LIN {X 0,Y 333.998,Z 557.276,A -85,B 0,C 180,E1 -14992.015,E2 -14992.015} C_VEL
LIN {X 0,Y 332.207,Z 566.269,A -85,B 0,C 180,E1 -14993.677,E2 -14993.677} C_VEL
LIN {X 0,Y 330.337,Z 575.114,A -85,B 0,C 180,E1 -14995.668,E2 -14995.668} C_VEL
LIN {X 0,Y 328.785,Z 582.446,A -85,B 0,C 180,E1 -14997.699,E2 -14997.699} C_VEL
LIN {X 0,Y 327.528,Z 588.358,A -85,B 0,C 180,E1 -14999.72,E2 -14999.72} C_VEL
LIN {X 0,Y 326.509,Z 593.499,A -85,B 0,C 180,E1 -15001.946,E2 -15001.946} C_VEL
LIN {X 0,Y 325.663,Z 597.746,A -85,B 0,C 180,E1 -15004.432,E2 -15004.432} C_VEL
LIN {X 0,Y 325.36,Z 599.436,A -85,B 0,C 180,E1 -15005.771,E2 -15005.771} C_VEL
LIN {X 0,Y 324.926,Z 601.645,A -85,B 0,C 180,E1 -15008.444,E2 -15008.444} C_VEL
LIN {X 0,Y 324.723,Z 602.327,A -85,B 0,C 180,E1 -15011.057,E2 -15011.057} C_VEL
LIN {X 0,Y 324.747,Z 602.109,A -85,B 0,C 180,E1 -15012.365,E2 -15012.365} C_VEL
LIN {X 0,Y 324.745,Z 600.606,A -85,B 0,C 180,E1 -15014.949,E2 -15014.949} C_VEL
LIN {X 0,Y 325.058,Z 597.666,A -85,B 0,C 180,E1 -15017.515,E2 -15017.515} C_VEL
LIN {X 0,Y 325.406,Z 594.514,A -85,B 0,C 180,E1 -15019.423,E2 -15019.423} C_VEL
LIN {X 0,Y 325.864,Z 590.445,A -85,B 0,C 180,E1 -15021.318,E2 -15021.318} C_VEL
LIN {X 0,Y 326.483,Z 585.399,A -85,B 0,C 180,E1 -15023.202,E2 -15023.202} C_VEL
LIN {X 0,Y 327.381,Z 578.186,A -85,B 0,C 180,E1 -15025.384,E2 -15025.384} C_VEL
LIN {X 0,Y 328.481,Z 570.619,A -85,B 0,C 180,E1 -15027.242,E2 -15027.242} C_VEL
LIN {X 0,Y 329.808,Z 561.53,A -85,B 0,C 180,E1 -15029.086,E2 -15029.086} C_VEL
LIN {X 0,Y 331.23,Z 550.578,A -85,B 0,C 180,E1 -15030.913,E2 -15030.913} C_VEL
LIN {X 0,Y 332.772,Z 539.376,A -85,B 0,C 180,E1 -15032.422,E2 -15032.422} C_VEL
LIN {X 0,Y 334.246,Z 527.017,A -85,B 0,C 180,E1 -15033.769,E2 -15033.769} C_VEL
LIN {X 0,Y 335.513,Z 515.129,A -85,B 0,C 180,E1 -15034.807,E2 -15034.807} C_VEL
LIN {X 0,Y 336.587,Z 502.215,A -85,B 0,C 180,E1 -15035.693,E2 -15035.693} C_VEL
LIN {X 0,Y 337.44,Z 488.43,A -85,B 0,C 180,E1 -15036.391,E2 -15036.391} C_VEL
LIN {X 0,Y 338.127,Z 474.079,A -85,B 0,C 180,E1 -15036.865,E2 -15036.865} C_VEL
LIN {X 0,Y 340.58,Z 375.262,A -85,B 0,C 180,E1 -15038.967,E2 -15038.967} C_VEL
LIN {X 0,Y 332.198,Z 352.897,A -85,B 0,C 180,E1 -15040.107,E2 -15040.107} C_VEL
LIN {X 0,Y 327.382,Z 341.262,A -85,B 0,C 180,E1 -15040.775,E2 -15040.775} C_VEL
LIN {X 0,Y 326.76,Z 338.405,A -85,B 0,C 180,E1 -15041.634,E2 -15041.634} C_VEL
LIN {X 0,Y 326.749,Z 338.41,A -85,B 0,C 180,E1 -15044.959,E2 -15044.959} C_VEL
LIN {X 0,Y 326.706,Z 338.416,A -85,B 0,C 180,E1 -15048.826,E2 -15048.826} C_VEL
LIN {X 0,Y 326.592,Z 338.429,A -85,B 0,C 180,E1 -15052.846,E2 -15052.846} C_VEL
LIN {X 0,Y 325.897,Z 338.513,A -85,B 0,C 180,E1 -15053.875,E2 -15053.875} C_VEL
LIN {X 0,Y 323.013,Z 338.873,A -85,B 0,C 180,E1 -15055.55,E2 -15055.55} C_VEL
LIN {X 0,Y 320.611,Z 339.175,A -85,B 0,C 180,E1 -15056.908,E2 -15056.908} C_VEL
LIN {X 0,Y 319.621,Z 339.294,A -85,B 0,C 180,E1 -15057.959,E2 -15057.959} C_VEL
LIN {X 0,Y 319.561,Z 339.302,A -85,B 0,C 180,E1 -15058.314,E2 -15058.314} C_VEL
LIN {X 0,Y 319.519,Z 339.306,A -85,B 0,C 180,E1 -15061.864,E2 -15061.864} C_VEL
LIN {X 0,Y 319.577,Z 339.297,A -85,B 0,C 180,E1 -15065.543,E2 -15065.543} C_VEL
LIN {X 0,Y 319.528,Z 339.306,A -85,B 0,C 180,E1 -15069.663,E2 -15069.663} C_VEL
LIN {X 0,Y 319.518,Z 339.302,A -85,B 0,C 180,E1 -15073.461,E2 -15073.461} C_VEL
LIN {X 0,Y 319.55,Z 339.304,A -85,B 0,C 180,E1 -15077.017,E2 -15077.017} C_VEL
LIN {X 0,Y 319.531,Z 339.307,A -85,B 0,C 180,E1 -15080.369,E2 -15080.369} C_VEL
LIN {X 0,Y 319.58,Z 339.294,A -85,B 0,C 180,E1 -15084.458,E2 -15084.458} C_VEL
LIN {X 0,Y 319.525,Z 339.307,A -85,B 0,C 180,E1 -15088.138,E2 -15088.138} C_VEL
LIN {X 0,Y 319.546,Z 339.302,A -85,B 0,C 180,E1 -15091.613,E2 -15091.613} C_VEL
LIN {X 0,Y 319.526,Z 339.306,A -85,B 0,C 180,E1 -15095.298,E2 -15095.298} C_VEL
LIN {X 0,Y 319.565,Z 339.302,A -85,B 0,C 180,E1 -15098.046,E2 -15098.046} C_VEL
LIN {X 0,Y 319.602,Z 339.299,A -85,B 0,C 180,E1 -15102.07,E2 -15102.07} C_VEL
LIN {X 0,Y 319.712,Z 339.281,A -85,B 0,C 180,E1 -15106.007,E2 -15106.007} C_VEL
LIN {X 0,Y 319.739,Z 339.276,A -85,B 0,C 180,E1 -15109.873,E2 -15109.873} C_VEL
LIN {X 0,Y 319.905,Z 339.26,A -85,B 0,C 180,E1 -15113.694,E2 -15113.694} C_VEL
LIN {X 0,Y 319.982,Z 339.246,A -85,B 0,C 180,E1 -15117.483,E2 -15117.483} C_VEL
LIN {X 0,Y 320.098,Z 339.23,A -85,B 0,C 180,E1 -15120,E2 -15120} C_VEL
LIN {X 0,Y 319.966,Z 339.25,A -85,B 0,C 180,E1 -15122.518,E2 -15122.518} C_VEL
LIN {X 0,Y 319.914,Z 339.259,A -85,B 0,C 180,E1 -15126.307,E2 -15126.307} C_VEL
LIN {X 0,Y 319.74,Z 339.282,A -85,B 0,C 180,E1 -15130.128,E2 -15130.128} C_VEL
LIN {X 0,Y 319.737,Z 339.282,A -85,B 0,C 180,E1 -15133.992,E2 -15133.992} C_VEL
LIN {X 0,Y 319.663,Z 339.291,A -85,B 0,C 180,E1 -15137.927,E2 -15137.927} C_VEL
LIN {X 0,Y 319.618,Z 339.293,A -85,B 0,C 180,E1 -15140.599,E2 -15140.599} C_VEL
LIN {X 0,Y 319.575,Z 339.302,A -85,B 0,C 180,E1 -15143.319,E2 -15143.319} C_VEL
LIN {X 0,Y 319.639,Z 339.292,A -85,B 0,C 180,E1 -15146.088,E2 -15146.088} C_VEL
LIN {X 0,Y 319.584,Z 339.298,A -85,B 0,C 180,E1 -15148.935,E2 -15148.935} C_VEL
LIN {X 0,Y 319.535,Z 339.306,A -85,B 0,C 180,E1 -15151.862,E2 -15151.862} C_VEL
LIN {X 0,Y 319.585,Z 339.302,A -85,B 0,C 180,E1 -15155.543,E2 -15155.543} C_VEL
LIN {X 0,Y 319.563,Z 339.304,A -85,B 0,C 180,E1 -15159.668,E2 -15159.668} C_VEL
LIN {X 0,Y 319.561,Z 339.305,A -85,B 0,C 180,E1 -15163.467,E2 -15163.467} C_VEL
LIN {X 0,Y 319.566,Z 339.303,A -85,B 0,C 180,E1 -15167.017,E2 -15167.017} C_VEL
LIN {X 0,Y 319.551,Z 339.304,A -85,B 0,C 180,E1 -15170.37,E2 -15170.37} C_VEL
LIN {X 0,Y 319.563,Z 339.306,A -85,B 0,C 180,E1 -15173.572,E2 -15173.572} C_VEL
LIN {X 0,Y 319.591,Z 339.4,A -85,B 0,C 180,E1 -15174.834,E2 -15174.834} C_VEL
LIN {X 0,Y 322.746,Z 352.977,A -85,B 0,C 180,E1 -15178.491,E2 -15178.491} C_VEL
LIN {X 0,Y 324.866,Z 363.071,A -85,B 0,C 180,E1 -15181.042,E2 -15181.042} C_VEL
LIN {X 0,Y 327.393,Z 370.408,A -85,B 0,C 180,E1 -15181.415,E2 -15181.415} C_VEL
LIN {X 0,Y 333.386,Z 408.912,A -85,B 0,C 180,E1 -15182.776,E2 -15182.776} C_VEL
LIN {X 0,Y 331.03,Z 501.06,A -85,B 0,C 180,E1 -15184.789,E2 -15184.789} C_VEL
LIN {X 0,Y 330.178,Z 515.8,A -85,B 0,C 180,E1 -15185.35,E2 -15185.35} C_VEL
LIN {X 0,Y 328.916,Z 529.85,A -85,B 0,C 180,E1 -15186.13,E2 -15186.13} C_VEL
LIN {X 0,Y 327.555,Z 542.941,A -85,B 0,C 180,E1 -15187.114,E2 -15187.114} C_VEL
LIN {X 0,Y 326.163,Z 555.029,A -85,B 0,C 180,E1 -15188.273,E2 -15188.273} C_VEL
LIN {X 0,Y 324.648,Z 566.029,A -85,B 0,C 180,E1 -15189.568,E2 -15189.568} C_VEL
LIN {X 0,Y 323.177,Z 575.846,A -85,B 0,C 180,E1 -15190.961,E2 -15190.961} C_VEL
LIN {X 0,Y 321.631,Z 586.724,A -85,B 0,C 180,E1 -15192.842,E2 -15192.842} C_VEL
LIN {X 0,Y 320.399,Z 595.692,A -85,B 0,C 180,E1 -15194.738,E2 -15194.738} C_VEL
LIN {X 0,Y 319.464,Z 603.139,A -85,B 0,C 180,E1 -15196.643,E2 -15196.643} C_VEL
LIN {X 0,Y 318.708,Z 609.322,A -85,B 0,C 180,E1 -15198.552,E2 -15198.552} C_VEL
LIN {X 0,Y 318.231,Z 614.435,A -85,B 0,C 180,E1 -15200.465,E2 -15200.465} C_VEL
LIN {X 0,Y 317.964,Z 619.684,A -85,B 0,C 180,E1 -15203.016,E2 -15203.016} C_VEL
LIN {X 0,Y 317.819,Z 622.616,A -85,B 0,C 180,E1 -15204.924,E2 -15204.924} C_VEL
LIN {X 0,Y 317.835,Z 624.104,A -85,B 0,C 180,E1 -15206.195,E2 -15206.195} C_VEL
LIN {X 0,Y 317.823,Z 626.005,A -85,B 0,C 180,E1 -15208.732,E2 -15208.732} C_VEL
LIN {X 0,Y 317.855,Z 626.441,A -85,B 0,C 180,E1 -15209.999,E2 -15209.999} C_VEL
LIN {X 0,Y 317.775,Z 626.296,A -85,B 0,C 180,E1 -15212.534,E2 -15212.534} C_VEL
LIN {X 0,Y 317.79,Z 624.814,A -85,B 0,C 180,E1 -15215.074,E2 -15215.074} C_VEL
LIN {X 0,Y 318.003,Z 621.974,A -85,B 0,C 180,E1 -15217.619,E2 -15217.619} C_VEL
LIN {X 0,Y 318.482,Z 617.709,A -85,B 0,C 180,E1 -15220.167,E2 -15220.167} C_VEL
LIN {X 0,Y 319.466,Z 611.91,A -85,B 0,C 180,E1 -15222.707,E2 -15222.707} C_VEL
LIN {X 0,Y 320.687,Z 605.414,A -85,B 0,C 180,E1 -15224.921,E2 -15224.921} C_VEL
LIN {X 0,Y 322.245,Z 597.392,A -85,B 0,C 180,E1 -15227.122,E2 -15227.122} C_VEL
LIN {X 0,Y 324.036,Z 589.033,A -85,B 0,C 180,E1 -15228.984,E2 -15228.984} C_VEL
LIN {X 0,Y 326.243,Z 579.004,A -85,B 0,C 180,E1 -15230.819,E2 -15230.819} C_VEL
LIN {X 0,Y 328.48,Z 567.861,A -85,B 0,C 180,E1 -15232.484,E2 -15232.484} C_VEL
LIN {X 0,Y 330.507,Z 556.826,A -85,B 0,C 180,E1 -15233.828,E2 -15233.828} C_VEL
LIN {X 0,Y 332.503,Z 544.873,A -85,B 0,C 180,E1 -15235.006,E2 -15235.006} C_VEL
LIN {X 0,Y 334.378,Z 531.726,A -85,B 0,C 180,E1 -15236.023,E2 -15236.023} C_VEL
LIN {X 0,Y 336.024,Z 518.149,A -85,B 0,C 180,E1 -15236.805,E2 -15236.805} C_VEL
LIN {X 0,Y 337.266,Z 504.224,A -85,B 0,C 180,E1 -15237.369,E2 -15237.369} C_VEL
LIN {X 0,Y 338.08,Z 485.357,A -85,B 0,C 180,E1 -15237.843,E2 -15237.843} C_VEL
LIN {X 0,Y 340.413,Z 409.919,A -85,B 0,C 180,E1 -15239.495,E2 -15239.495} C_VEL
LIN {X 0,Y 337.287,Z 391.526,A -85,B 0,C 180,E1 -15240.327,E2 -15240.327} C_VEL
LIN {X 0,Y 335.087,Z 381.47,A -85,B 0,C 180,E1 -15240.852,E2 -15240.852} C_VEL
LIN {X 0,Y 327.611,Z 365.686,A -85,B 0,C 180,E1 -15242.225,E2 -15242.225} C_VEL
LIN {X 0,Y 325.569,Z 361.41,A -85,B 0,C 180,E1 -15242.66,E2 -15242.66} C_VEL
LIN {X 0,Y 323.248,Z 352.03,A -85,B 0,C 180,E1 -15245.561,E2 -15245.561} C_VEL
LIN {X 0,Y 320.051,Z 341.028,A -85,B 0,C 180,E1 -15249.281,E2 -15249.281} C_VEL
LIN {X 0,Y 319.58,Z 339.301,A -85,B 0,C 180,E1 -15249.919,E2 -15249.919} C_VEL
LIN {X 0,Y 319.558,Z 339.305,A -85,B 0,C 180,E1 -15253.467,E2 -15253.467} C_VEL
LIN {X 0,Y 319.55,Z 339.297,A -85,B 0,C 180,E1 -15257.015,E2 -15257.015} C_VEL
LIN {X 0,Y 319.542,Z 339.286,A -85,B 0,C 180,E1 -15260.37,E2 -15260.37} C_VEL
LIN {X 0,Y 319.554,Z 339.304,A -85,B 0,C 180,E1 -15263.571,E2 -15263.571} C_VEL
LIN {X 0,Y 319.572,Z 339.298,A -85,B 0,C 180,E1 -15266.685,E2 -15266.685} C_VEL
LIN {X 0,Y 319.585,Z 339.298,A -85,B 0,C 180,E1 -15269.616,E2 -15269.616} C_VEL
LIN {X 0,Y 319.603,Z 339.296,A -85,B 0,C 180,E1 -15272.497,E2 -15272.497} C_VEL
LIN {X 0,Y 319.597,Z 339.299,A -85,B 0,C 180,E1 -15275.303,E2 -15275.303} C_VEL
LIN {X 0,Y 319.59,Z 339.295,A -85,B 0,C 180,E1 -15278.047,E2 -15278.047} C_VEL
LIN {X 0,Y 319.682,Z 339.279,A -85,B 0,C 180,E1 -15280.961,E2 -15280.961} C_VEL
LIN {X 0,Y 319.724,Z 339.274,A -85,B 0,C 180,E1 -15285.275,E2 -15285.275} C_VEL
LIN {X 0,Y 319.75,Z 339.274,A -85,B 0,C 180,E1 -15289.872,E2 -15289.872} C_VEL
LIN {X 0,Y 319.924,Z 339.251,A -85,B 0,C 180,E1 -15292.426,E2 -15292.426} C_VEL
LIN {X 0,Y 319.726,Z 339.283,A -85,B 0,C 180,E1 -15294.955,E2 -15294.955} C_VEL
LIN {X 0,Y 320.006,Z 339.247,A -85,B 0,C 180,E1 -15298.741,E2 -15298.741} C_VEL
LIN {X 0,Y 319.952,Z 339.254,A -85,B 0,C 180,E1 -15302.517,E2 -15302.517} C_VEL
LIN {X 0,Y 319.874,Z 339.263,A -85,B 0,C 180,E1 -15306.452,E2 -15306.452} C_VEL
LIN {X 0,Y 319.725,Z 339.282,A -85,B 0,C 180,E1 -15310.128,E2 -15310.128} C_VEL
LIN {X 0,Y 319.721,Z 339.285,A -85,B 0,C 180,E1 -15313.992,E2 -15313.992} C_VEL
LIN {X 0,Y 319.605,Z 339.299,A -85,B 0,C 180,E1 -15317.93,E2 -15317.93} C_VEL
LIN {X 0,Y 319.558,Z 339.299,A -85,B 0,C 180,E1 -15321.955,E2 -15321.955} C_VEL
LIN {X 0,Y 319.561,Z 339.306,A -85,B 0,C 180,E1 -15326.094,E2 -15326.094} C_VEL
LIN {X 0,Y 319.534,Z 339.292,A -85,B 0,C 180,E1 -15328.939,E2 -15328.939} C_VEL
LIN {X 0,Y 319.515,Z 339.308,A -85,B 0,C 180,E1 -15331.863,E2 -15331.863} C_VEL
LIN {X 0,Y 319.571,Z 339.303,A -85,B 0,C 180,E1 -15335.543,E2 -15335.543} C_VEL
LIN {X 0,Y 319.617,Z 339.487,A -85,B 0,C 180,E1 -15337.426,E2 -15337.426} C_VEL
LIN {X 0,Y 320.649,Z 343.22,A -85,B 0,C 180,E1 -15338.757,E2 -15338.757} C_VEL
LIN {X 0,Y 329.908,Z 359.392,A -85,B 0,C 180,E1 -15340.471,E2 -15340.471} C_VEL
LIN {X 0,Y 338.34,Z 376.267,A -85,B 0,C 180,E1 -15341.968,E2 -15341.968} C_VEL
LIN {X 0,Y 341.303,Z 383.071,A -85,B 0,C 180,E1 -15342.489,E2 -15342.489} C_VEL
LIN {X 0,Y 338.045,Z 478.993,A -85,B 0,C 180,E1 -15344.599,E2 -15344.599} C_VEL
LIN {X 0,Y 337.093,Z 493.304,A -85,B 0,C 180,E1 -15345.152,E2 -15345.152} C_VEL
LIN {X 0,Y 335.699,Z 507.187,A -85,B 0,C 180,E1 -15345.928,E2 -15345.928} C_VEL
LIN {X 0,Y 334.177,Z 519.863,A -85,B 0,C 180,E1 -15346.884,E2 -15346.884} C_VEL
LIN {X 0,Y 332.33,Z 531.906,A -85,B 0,C 180,E1 -15348.028,E2 -15348.028} C_VEL
LIN {X 0,Y 330.115,Z 544.38,A -85,B 0,C 180,E1 -15349.511,E2 -15349.511} C_VEL
LIN {X 0,Y 328.147,Z 554.61,A -85,B 0,C 180,E1 -15351.016,E2 -15351.016} C_VEL
LIN {X 0,Y 325.919,Z 565.245,A -85,B 0,C 180,E1 -15352.925,E2 -15352.925} C_VEL
LIN {X 0,Y 323.915,Z 574.161,A -85,B 0,C 180,E1 -15354.904,E2 -15354.904} C_VEL
LIN {X 0,Y 322.226,Z 581.674,A -85,B 0,C 180,E1 -15356.959,E2 -15356.959} C_VEL
LIN {X 0,Y 320.777,Z 588.147,A -85,B 0,C 180,E1 -15359.16,E2 -15359.16} C_VEL
LIN {X 0,Y 319.568,Z 593.725,A -85,B 0,C 180,E1 -15361.603,E2 -15361.603} C_VEL
LIN {X 0,Y 318.764,Z 597.561,A -85,B 0,C 180,E1 -15363.837,E2 -15363.837} C_VEL
LIN {X 0,Y 318.381,Z 599.336,A -85,B 0,C 180,E1 -15365.204,E2 -15365.204} C_VEL
LIN {X 0,Y 317.881,Z 601.705,A -85,B 0,C 180,E1 -15367.925,E2 -15367.925} C_VEL
LIN {X 0,Y 317.66,Z 602.572,A -85,B 0,C 180,E1 -15370.619,E2 -15370.619} C_VEL
LIN {X 0,Y 317.635,Z 601.988,A -85,B 0,C 180,E1 -15373.285,E2 -15373.285} C_VEL
LIN {X 0,Y 317.724,Z 599.958,A -85,B 0,C 180,E1 -15375.919,E2 -15375.919} C_VEL
LIN {X 0,Y 318.167,Z 596.446,A -85,B 0,C 180,E1 -15378.534,E2 -15378.534} C_VEL
LIN {X 0,Y 318.714,Z 591.422,A -85,B 0,C 180,E1 -15381.122,E2 -15381.122} C_VEL
LIN {X 0,Y 319.361,Z 586.558,A -85,B 0,C 180,E1 -15383.049,E2 -15383.049} C_VEL
LIN {X 0,Y 320.242,Z 579.551,A -85,B 0,C 180,E1 -15385.281,E2 -15385.281} C_VEL
LIN {X 0,Y 321.52,Z 570.855,A -85,B 0,C 180,E1 -15387.496,E2 -15387.496} C_VEL
LIN {X 0,Y 322.906,Z 561.75,A -85,B 0,C 180,E1 -15389.378,E2 -15389.378} C_VEL
LIN {X 0,Y 324.139,Z 552.572,A -85,B 0,C 180,E1 -15390.959,E2 -15390.959} C_VEL
LIN {X 0,Y 325.696,Z 541.915,A -85,B 0,C 180,E1 -15392.475,E2 -15392.475} C_VEL
LIN {X 0,Y 327.149,Z 530.134,A -85,B 0,C 180,E1 -15393.85,E2 -15393.85} C_VEL
LIN {X 0,Y 328.631,Z 517.116,A -85,B 0,C 180,E1 -15395.062,E2 -15395.062} C_VEL
LIN {X 0,Y 329.818,Z 503.556,A -85,B 0,C 180,E1 -15396.04,E2 -15396.04} C_VEL
LIN {X 0,Y 330.775,Z 489.268,A -85,B 0,C 180,E1 -15396.789,E2 -15396.789} C_VEL
LIN {X 0,Y 331.485,Z 475.269,A -85,B 0,C 180,E1 -15397.271,E2 -15397.271} C_VEL
LIN {X 0,Y 334.019,Z 376.85,A -85,B 0,C 180,E1 -15399.406,E2 -15399.406} C_VEL
LIN {X 0,Y 326.131,Z 355.83,A -85,B 0,C 180,E1 -15400.512,E2 -15400.512} C_VEL
LIN {X 0,Y 320.207,Z 341.543,A -85,B 0,C 180,E1 -15401.357,E2 -15401.357} C_VEL
LIN {X 0,Y 319.713,Z 339.283,A -85,B 0,C 180,E1 -15402.055,E2 -15402.055} C_VEL
LIN {X 0,Y 319.678,Z 339.293,A -85,B 0,C 180,E1 -15405.298,E2 -15405.298} C_VEL
LIN {X 0,Y 319.628,Z 339.3,A -85,B 0,C 180,E1 -15409.259,E2 -15409.259} C_VEL
LIN {X 0,Y 319.549,Z 339.307,A -85,B 0,C 180,E1 -15413.322,E2 -15413.322} C_VEL
LIN {X 0,Y 319.566,Z 339.301,A -85,B 0,C 180,E1 -15416.095,E2 -15416.095} C_VEL
LIN {X 0,Y 319.561,Z 339.302,A -85,B 0,C 180,E1 -15418.314,E2 -15418.314} C_VEL
LIN {X 0,Y 318.95,Z 339.382,A -85,B 0,C 180,E1 -15419.365,E2 -15419.365} C_VEL
LIN {X 0,Y 316.115,Z 339.735,A -85,B 0,C 180,E1 -15421.076,E2 -15421.076} C_VEL
LIN {X 0,Y 313.668,Z 340.038,A -85,B 0,C 180,E1 -15422.462,E2 -15422.462} C_VEL
LIN {X 0,Y 312.603,Z 340.17,A -85,B 0,C 180,E1 -15423.536,E2 -15423.536} C_VEL
LIN {X 0,Y 312.51,Z 340.18,A -85,B 0,C 180,E1 -15423.9,E2 -15423.9} C_VEL
LIN {X 0,Y 312.512,Z 340.178,A -85,B 0,C 180,E1 -15427.388,E2 -15427.388} C_VEL
LIN {X 0,Y 312.44,Z 340.193,A -85,B 0,C 180,E1 -15430.718,E2 -15430.718} C_VEL
LIN {X 0,Y 312.45,Z 340.182,A -85,B 0,C 180,E1 -15434.211,E2 -15434.211} C_VEL
LIN {X 0,Y 312.454,Z 340.186,A -85,B 0,C 180,E1 -15437.926,E2 -15437.926} C_VEL
LIN {X 0,Y 312.476,Z 340.181,A -85,B 0,C 180,E1 -15441.925,E2 -15441.925} C_VEL
LIN {X 0,Y 312.531,Z 340.169,A -85,B 0,C 180,E1 -15444.221,E2 -15444.221} C_VEL
LIN {X 0,Y 312.503,Z 340.179,A -85,B 0,C 180,E1 -15447.334,E2 -15447.334} C_VEL
LIN {X 0,Y 312.487,Z 340.181,A -85,B 0,C 180,E1 -15451.3,E2 -15451.3} C_VEL
LIN {X 0,Y 312.517,Z 340.182,A -85,B 0,C 180,E1 -15454.706,E2 -15454.706} C_VEL
LIN {X 0,Y 312.541,Z 340.174,A -85,B 0,C 180,E1 -15457.526,E2 -15457.526} C_VEL
LIN {X 0,Y 312.561,Z 340.174,A -85,B 0,C 180,E1 -15461.652,E2 -15461.652} C_VEL
LIN {X 0,Y 312.654,Z 340.158,A -85,B 0,C 180,E1 -15465.685,E2 -15465.685} C_VEL
LIN {X 0,Y 312.689,Z 340.152,A -85,B 0,C 180,E1 -15469.642,E2 -15469.642} C_VEL
LIN {X 0,Y 312.8,Z 340.147,A -85,B 0,C 180,E1 -15472.253,E2 -15472.253} C_VEL
LIN {X 0,Y 312.701,Z 340.155,A -85,B 0,C 180,E1 -15474.843,E2 -15474.843} C_VEL
LIN {X 0,Y 312.985,Z 340.111,A -85,B 0,C 180,E1 -15478.714,E2 -15478.714} C_VEL
LIN {X 0,Y 312.986,Z 340.114,A -85,B 0,C 180,E1 -15481.287,E2 -15481.287} C_VEL
LIN {X 0,Y 312.857,Z 340.137,A -85,B 0,C 180,E1 -15486.449,E2 -15486.449} C_VEL
LIN {X 0,Y 312.755,Z 340.147,A -85,B 0,C 180,E1 -15489.051,E2 -15489.051} C_VEL
LIN {X 0,Y 312.638,Z 340.163,A -85,B 0,C 180,E1 -15492.991,E2 -15492.991} C_VEL
LIN {X 0,Y 312.643,Z 340.167,A -85,B 0,C 180,E1 -15495.65,E2 -15495.65} C_VEL
LIN {X 0,Y 312.635,Z 340.164,A -85,B 0,C 180,E1 -15499.236,E2 -15499.236} C_VEL
LIN {X 0,Y 312.551,Z 340.174,A -85,B 0,C 180,E1 -15502.789,E2 -15502.789} C_VEL
LIN {X 0,Y 312.607,Z 340.169,A -85,B 0,C 180,E1 -15505.935,E2 -15505.935} C_VEL
LIN {X 0,Y 312.543,Z 340.178,A -85,B 0,C 180,E1 -15509.651,E2 -15509.651} C_VEL
LIN {X 0,Y 312.524,Z 340.181,A -85,B 0,C 180,E1 -15513.689,E2 -15513.689} C_VEL
LIN {X 0,Y 312.526,Z 340.178,A -85,B 0,C 180,E1 -15517.386,E2 -15517.386} C_VEL
LIN {X 0,Y 312.495,Z 340.183,A -85,B 0,C 180,E1 -15520.709,E2 -15520.709} C_VEL
LIN {X 0,Y 312.477,Z 340.184,A -85,B 0,C 180,E1 -15524.206,E2 -15524.206} C_VEL
LIN {X 0,Y 312.49,Z 340.184,A -85,B 0,C 180,E1 -15527.918,E2 -15527.918} C_VEL
LIN {X 0,Y 312.51,Z 340.182,A -85,B 0,C 180,E1 -15531.917,E2 -15531.917} C_VEL
LIN {X 0,Y 312.55,Z 340.271,A -85,B 0,C 180,E1 -15534.371,E2 -15534.371} C_VEL
LIN {X 0,Y 315.436,Z 352.83,A -85,B 0,C 180,E1 -15537.85,E2 -15537.85} C_VEL
LIN {X 0,Y 317.594,Z 362.843,A -85,B 0,C 180,E1 -15540.447,E2 -15540.447} C_VEL
LIN {X 0,Y 321.015,Z 372.074,A -85,B 0,C 180,E1 -15540.954,E2 -15540.954} C_VEL
LIN {X 0,Y 326.806,Z 410.08,A -85,B 0,C 180,E1 -15542.322,E2 -15542.322} C_VEL
LIN {X 0,Y 324.386,Z 501.432,A -85,B 0,C 180,E1 -15544.364,E2 -15544.364} C_VEL
LIN {X 0,Y 323.509,Z 515.953,A -85,B 0,C 180,E1 -15544.935,E2 -15544.935} C_VEL
LIN {X 0,Y 322.149,Z 530.463,A -85,B 0,C 180,E1 -15545.768,E2 -15545.768} C_VEL
LIN {X 0,Y 320.617,Z 544.514,A -85,B 0,C 180,E1 -15546.87,E2 -15546.87} C_VEL
LIN {X 0,Y 319.239,Z 555.943,A -85,B 0,C 180,E1 -15548.021,E2 -15548.021} C_VEL
LIN {X 0,Y 317.567,Z 567.413,A -85,B 0,C 180,E1 -15549.431,E2 -15549.431} C_VEL
LIN {X 0,Y 316.095,Z 576.961,A -85,B 0,C 180,E1 -15550.855,E2 -15550.855} C_VEL
LIN {X 0,Y 314.544,Z 587.62,A -85,B 0,C 180,E1 -15552.778,E2 -15552.778} C_VEL
LIN {X 0,Y 313.275,Z 596.432,A -85,B 0,C 180,E1 -15554.723,E2 -15554.723} C_VEL
LIN {X 0,Y 312.513,Z 602.546,A -85,B 0,C 180,E1 -15556.341,E2 -15556.341} C_VEL
LIN {X 0,Y 311.713,Z 608.794,A -85,B 0,C 180,E1 -15558.291,E2 -15558.291} C_VEL
LIN {X 0,Y 311.195,Z 613.958,A -85,B 0,C 180,E1 -15560.247,E2 -15560.247} C_VEL
LIN {X 0,Y 310.89,Z 619.266,A -85,B 0,C 180,E1 -15562.857,E2 -15562.857} C_VEL
LIN {X 0,Y 310.725,Z 622.222,A -85,B 0,C 180,E1 -15564.808,E2 -15564.808} C_VEL
LIN {X 0,Y 310.744,Z 623.738,A -85,B 0,C 180,E1 -15566.108,E2 -15566.108} C_VEL
LIN {X 0,Y 310.733,Z 625.697,A -85,B 0,C 180,E1 -15568.703,E2 -15568.703} C_VEL
LIN {X 0,Y 310.762,Z 626.158,A -85,B 0,C 180,E1 -15569.999,E2 -15569.999} C_VEL
LIN {X 0,Y 310.697,Z 626.059,A -85,B 0,C 180,E1 -15572.592,E2 -15572.592} C_VEL
LIN {X 0,Y 310.696,Z 624.622,A -85,B 0,C 180,E1 -15575.19,E2 -15575.19} C_VEL
LIN {X 0,Y 310.949,Z 621.834,A -85,B 0,C 180,E1 -15577.793,E2 -15577.793} C_VEL
LIN {X 0,Y 311.46,Z 617.623,A -85,B 0,C 180,E1 -15580.399,E2 -15580.399} C_VEL
LIN {X 0,Y 312.505,Z 611.878,A -85,B 0,C 180,E1 -15582.995,E2 -15582.995} C_VEL
LIN {X 0,Y 313.795,Z 605.442,A -85,B 0,C 180,E1 -15585.256,E2 -15585.256} C_VEL
LIN {X 0,Y 315.441,Z 597.486,A -85,B 0,C 180,E1 -15587.503,E2 -15587.503} C_VEL
LIN {X 0,Y 317.321,Z 589.201,A -85,B 0,C 180,E1 -15589.402,E2 -15589.402} C_VEL
LIN {X 0,Y 319.605,Z 579.27,A -85,B 0,C 180,E1 -15591.273,E2 -15591.273} C_VEL
LIN {X 0,Y 321.948,Z 568.274,A -85,B 0,C 180,E1 -15592.966,E2 -15592.966} C_VEL
LIN {X 0,Y 324.299,Z 556.189,A -85,B 0,C 180,E1 -15594.467,E2 -15594.467} C_VEL
LIN {X 0,Y 326.42,Z 543.986,A -85,B 0,C 180,E1 -15595.676,E2 -15595.676} C_VEL
LIN {X 0,Y 328.38,Z 530.665,A -85,B 0,C 180,E1 -15596.706,E2 -15596.706} C_VEL
LIN {X 0,Y 330.163,Z 516.07,A -85,B 0,C 180,E1 -15597.535,E2 -15597.535} C_VEL
LIN {X 0,Y 331.344,Z 502.398,A -85,B 0,C 180,E1 -15598.072,E2 -15598.072} C_VEL
LIN {X 0,Y 332.283,Z 479.275,A -85,B 0,C 180,E1 -15598.631,E2 -15598.631} C_VEL
LIN {X 0,Y 334.508,Z 411.118,A -85,B 0,C 180,E1 -15600.145,E2 -15600.145} C_VEL
LIN {X 0,Y 331.617,Z 393.689,A -85,B 0,C 180,E1 -15600.953,E2 -15600.953} C_VEL
LIN {X 0,Y 329.721,Z 384.75,A -85,B 0,C 180,E1 -15601.431,E2 -15601.431} C_VEL
LIN {X 0,Y 322.677,Z 369.761,A -85,B 0,C 180,E1 -15602.771,E2 -15602.771} C_VEL
LIN {X 0,Y 318.361,Z 361.182,A -85,B 0,C 180,E1 -15603.636,E2 -15603.636} C_VEL
LIN {X 0,Y 315.712,Z 351.035,A -85,B 0,C 180,E1 -15606.943,E2 -15606.943} C_VEL
LIN {X 0,Y 313.381,Z 343.26,A -85,B 0,C 180,E1 -15609.697,E2 -15609.697} C_VEL
LIN {X 0,Y 312.517,Z 340.177,A -85,B 0,C 180,E1 -15610.916,E2 -15610.916} C_VEL
LIN {X 0,Y 312.461,Z 340.189,A -85,B 0,C 180,E1 -15614.206,E2 -15614.206} C_VEL
LIN {X 0,Y 312.48,Z 340.187,A -85,B 0,C 180,E1 -15617.917,E2 -15617.917} C_VEL
LIN {X 0,Y 312.53,Z 340.173,A -85,B 0,C 180,E1 -15621.909,E2 -15621.909} C_VEL
LIN {X 0,Y 312.501,Z 340.184,A -85,B 0,C 180,E1 -15625.789,E2 -15625.789} C_VEL
LIN {X 0,Y 312.518,Z 340.181,A -85,B 0,C 180,E1 -15628.853,E2 -15628.853} C_VEL
LIN {X 0,Y 312.569,Z 340.175,A -85,B 0,C 180,E1 -15631.824,E2 -15631.824} C_VEL
LIN {X 0,Y 312.578,Z 340.172,A -85,B 0,C 180,E1 -15634.71,E2 -15634.71} C_VEL
LIN {X 0,Y 312.58,Z 340.164,A -85,B 0,C 180,E1 -15637.528,E2 -15637.528} C_VEL
LIN {X 0,Y 312.631,Z 340.159,A -85,B 0,C 180,E1 -15641.656,E2 -15641.656} C_VEL
LIN {X 0,Y 312.686,Z 340.152,A -85,B 0,C 180,E1 -15645.685,E2 -15645.685} C_VEL
LIN {X 0,Y 312.694,Z 340.15,A -85,B 0,C 180,E1 -15649.641,E2 -15649.641} C_VEL
LIN {X 0,Y 312.863,Z 340.131,A -85,B 0,C 180,E1 -15652.254,E2 -15652.254} C_VEL
LIN {X 0,Y 312.9,Z 340.124,A -85,B 0,C 180,E1 -15653.551,E2 -15653.551} C_VEL
LIN {X 0,Y 312.973,Z 340.124,A -85,B 0,C 180,E1 -15658.713,E2 -15658.713} C_VEL
LIN {X 0,Y 312.901,Z 340.132,A -85,B 0,C 180,E1 -15662.574,E2 -15662.574} C_VEL
LIN {X 0,Y 312.829,Z 340.141,A -85,B 0,C 180,E1 -15666.449,E2 -15666.449} C_VEL
LIN {X 0,Y 312.741,Z 340.146,A -85,B 0,C 180,E1 -15669.05,E2 -15669.05} C_VEL
LIN {X 0,Y 312.622,Z 340.161,A -85,B 0,C 180,E1 -15672.991,E2 -15672.991} C_VEL
LIN {X 0,Y 312.612,Z 340.164,A -85,B 0,C 180,E1 -15675.651,E2 -15675.651} C_VEL
LIN {X 0,Y 312.53,Z 340.176,A -85,B 0,C 180,E1 -15679.713,E2 -15679.713} C_VEL
LIN {X 0,Y 312.513,Z 340.177,A -85,B 0,C 180,E1 -15682.779,E2 -15682.779} C_VEL
LIN {X 0,Y 312.521,Z 340.184,A -85,B 0,C 180,E1 -15685.908,E2 -15685.908} C_VEL
LIN {X 0,Y 312.487,Z 340.175,A -85,B 0,C 180,E1 -15689.655,E2 -15689.655} C_VEL
LIN {X 0,Y 312.511,Z 340.175,A -85,B 0,C 180,E1 -15693.689,E2 -15693.689} C_VEL
LIN {X 0,Y 312.55,Z 340.329,A -85,B 0,C 180,E1 -15696.496,E2 -15696.496} C_VEL
LIN {X 0,Y 313.437,Z 343.461,A -85,B 0,C 180,E1 -15697.691,E2 -15697.691} C_VEL
LIN {X 0,Y 315.958,Z 347.622,A -85,B 0,C 180,E1 -15698.198,E2 -15698.198} C_VEL
LIN {X 0,Y 325.012,Z 363.494,A -85,B 0,C 180,E1 -15699.936,E2 -15699.936} C_VEL
LIN {X 0,Y 332.939,Z 379.491,A -85,B 0,C 180,E1 -15701.399,E2 -15701.399} C_VEL
LIN {X 0,Y 335.419,Z 385.177,A -85,B 0,C 180,E1 -15701.852,E2 -15701.852} C_VEL
LIN {X 0,Y 332.103,Z 478.68,A -85,B 0,C 180,E1 -15703.933,E2 -15703.933} C_VEL
LIN {X 0,Y 331.145,Z 492.897,A -85,B 0,C 180,E1 -15704.48,E2 -15704.48} C_VEL
LIN {X 0,Y 329.848,Z 505.59,A -85,B 0,C 180,E1 -15705.174,E2 -15705.174} C_VEL
LIN {X 0,Y 328.262,Z 518.459,A -85,B 0,C 180,E1 -15706.123,E2 -15706.123} C_VEL
LIN {X 0,Y 326.355,Z 530.793,A -85,B 0,C 180,E1 -15707.282,E2 -15707.282} C_VEL
LIN {X 0,Y 324.267,Z 542.27,A -85,B 0,C 180,E1 -15708.622,E2 -15708.622} C_VEL
LIN {X 0,Y 322.176,Z 552.531,A -85,B 0,C 180,E1 -15710.085,E2 -15710.085} C_VEL
LIN {X 0,Y 320.215,Z 561.791,A -85,B 0,C 180,E1 -15711.684,E2 -15711.684} C_VEL
LIN {X 0,Y 317.924,Z 571.595,A -85,B 0,C 180,E1 -15713.75,E2 -15713.75} C_VEL
LIN {X 0,Y 316.116,Z 579.17,A -85,B 0,C 180,E1 -15715.707,E2 -15715.707} C_VEL
LIN {X 0,Y 314.688,Z 585.204,A -85,B 0,C 180,E1 -15717.59,E2 -15717.59} C_VEL
LIN {X 0,Y 313.387,Z 590.687,A -85,B 0,C 180,E1 -15719.698,E2 -15719.698} C_VEL
LIN {X 0,Y 312.409,Z 595.013,A -85,B 0,C 180,E1 -15721.81,E2 -15721.81} C_VEL
LIN {X 0,Y 311.479,Z 599.096,A -85,B 0,C 180,E1 -15724.492,E2 -15724.492} C_VEL
LIN {X 0,Y 311.105,Z 600.707,A -85,B 0,C 180,E1 -15726.008,E2 -15726.008} C_VEL
LIN {X 0,Y 310.697,Z 602.479,A -85,B 0,C 180,E1 -15728.783,E2 -15728.783} C_VEL
LIN {X 0,Y 310.549,Z 602.776,A -85,B 0,C 180,E1 -15731.53,E2 -15731.53} C_VEL
LIN {X 0,Y 310.534,Z 601.64,A -85,B 0,C 180,E1 -15734.243,E2 -15734.243} C_VEL
LIN {X 0,Y 310.81,Z 599.076,A -85,B 0,C 180,E1 -15736.933,E2 -15736.933} C_VEL
LIN {X 0,Y 311.144,Z 596.148,A -85,B 0,C 180,E1 -15738.932,E2 -15738.932} C_VEL
LIN {X 0,Y 311.744,Z 590.936,A -85,B 0,C 180,E1 -15741.575,E2 -15741.575} C_VEL
LIN {X 0,Y 312.4,Z 585.878,A -85,B 0,C 180,E1 -15743.543,E2 -15743.543} C_VEL
LIN {X 0,Y 313.403,Z 578.642,A -85,B 0,C 180,E1 -15745.822,E2 -15745.822} C_VEL
LIN {X 0,Y 314.583,Z 571.053,A -85,B 0,C 180,E1 -15747.761,E2 -15747.761} C_VEL
LIN {X 0,Y 316.001,Z 561.941,A -85,B 0,C 180,E1 -15749.683,E2 -15749.683} C_VEL
LIN {X 0,Y 317.262,Z 552.907,A -85,B 0,C 180,E1 -15751.27,E2 -15751.27} C_VEL
LIN {X 0,Y 318.905,Z 542.063,A -85,B 0,C 180,E1 -15752.843,E2 -15752.843} C_VEL
LIN {X 0,Y 320.433,Z 530.247,A -85,B 0,C 180,E1 -15754.246,E2 -15754.246} C_VEL
LIN {X 0,Y 321.938,Z 517.207,A -85,B 0,C 180,E1 -15755.482,E2 -15755.482} C_VEL
LIN {X 0,Y 323.18,Z 503.562,A -85,B 0,C 180,E1 -15756.478,E2 -15756.478} C_VEL
LIN {X 0,Y 324.18,Z 489.154,A -85,B 0,C 180,E1 -15757.24,E2 -15757.24} C_VEL
LIN {X 0,Y 324.901,Z 474.939,A -85,B 0,C 180,E1 -15757.732,E2 -15757.732} C_VEL
LIN {X 0,Y 327.513,Z 378.63,A -85,B 0,C 180,E1 -15759.855,E2 -15759.855} C_VEL
LIN {X 0,Y 320.314,Z 359.232,A -85,B 0,C 180,E1 -15760.9,E2 -15760.9} C_VEL
LIN {X 0,Y 313.014,Z 341.738,A -85,B 0,C 180,E1 -15761.988,E2 -15761.988} C_VEL
LIN {X 0,Y 312.647,Z 340.164,A -85,B 0,C 180,E1 -15762.496,E2 -15762.496} C_VEL
LIN {X 0,Y 312.621,Z 340.171,A -85,B 0,C 180,E1 -15765.652,E2 -15765.652} C_VEL
LIN {X 0,Y 312.559,Z 340.178,A -85,B 0,C 180,E1 -15769.712,E2 -15769.712} C_VEL
LIN {X 0,Y 312.52,Z 340.183,A -85,B 0,C 180,E1 -15772.779,E2 -15772.779} C_VEL
LIN {X 0,Y 312.527,Z 340.178,A -85,B 0,C 180,E1 -15775.908,E2 -15775.908} C_VEL
LIN {X 0,Y 312.47,Z 340.186,A -85,B 0,C 180,E1 -15779.659,E2 -15779.659} C_VEL
LIN {X 0,Y 312.519,Z 340.179,A -85,B 0,C 180,E1 -15783.69,E2 -15783.69} C_VEL
LIN {X 0,Y 312.51,Z 340.18,A -85,B 0,C 180,E1 -15783.9,E2 -15783.9} C_VEL
LIN {X 0,Y 311.818,Z 340.268,A -85,B 0,C 180,E1 -15784.974,E2 -15784.974} C_VEL
LIN {X 0,Y 308.929,Z 340.624,A -85,B 0,C 180,E1 -15786.723,E2 -15786.723} C_VEL
LIN {X 0,Y 306.499,Z 340.926,A -85,B 0,C 180,E1 -15788.14,E2 -15788.14} C_VEL
LIN {X 0,Y 305.469,Z 341.059,A -85,B 0,C 180,E1 -15789.239,E2 -15789.239} C_VEL
LIN {X 0,Y 305.391,Z 341.064,A -85,B 0,C 180,E1 -15789.611,E2 -15789.611} C_VEL
LIN {X 0,Y 305.42,Z 341.056,A -85,B 0,C 180,E1 -15793.657,E2 -15793.657} C_VEL
LIN {X 0,Y 305.434,Z 341.06,A -85,B 0,C 180,E1 -15797.42,E2 -15797.42} C_VEL
LIN {X 0,Y 305.445,Z 341.056,A -85,B 0,C 180,E1 -15801.594,E2 -15801.594} C_VEL
LIN {X 0,Y 305.463,Z 341.053,A -85,B 0,C 180,E1 -15804.888,E2 -15804.888} C_VEL
LIN {X 0,Y 305.443,Z 341.062,A -85,B 0,C 180,E1 -15808.359,E2 -15808.359} C_VEL
LIN {X 0,Y 305.455,Z 341.058,A -85,B 0,C 180,E1 -15811.108,E2 -15811.108} C_VEL
LIN {X 0,Y 305.48,Z 341.056,A -85,B 0,C 180,E1 -15814.08,E2 -15814.08} C_VEL
LIN {X 0,Y 305.462,Z 341.059,A -85,B 0,C 180,E1 -15818.401,E2 -15818.401} C_VEL
LIN {X 0,Y 305.515,Z 341.051,A -85,B 0,C 180,E1 -15821.213,E2 -15821.213} C_VEL
LIN {X 0,Y 305.582,Z 341.037,A -85,B 0,C 180,E1 -15825.346,E2 -15825.346} C_VEL
LIN {X 0,Y 305.627,Z 341.029,A -85,B 0,C 180,E1 -15829.4,E2 -15829.4} C_VEL
LIN {X 0,Y 305.75,Z 341.024,A -85,B 0,C 180,E1 -15832.073,E2 -15832.073} C_VEL
LIN {X 0,Y 305.67,Z 341.031,A -85,B 0,C 180,E1 -15834.724,E2 -15834.724} C_VEL
LIN {X 0,Y 305.953,Z 340.986,A -85,B 0,C 180,E1 -15838.684,E2 -15838.684} C_VEL
LIN {X 0,Y 305.953,Z 340.989,A -85,B 0,C 180,E1 -15841.317,E2 -15841.317} C_VEL
LIN {X 0,Y 305.803,Z 341.015,A -85,B 0,C 180,E1 -15846.599,E2 -15846.599} C_VEL
LIN {X 0,Y 305.699,Z 341.027,A -85,B 0,C 180,E1 -15849.261,E2 -15849.261} C_VEL
LIN {X 0,Y 305.593,Z 341.042,A -85,B 0,C 180,E1 -15853.296,E2 -15853.296} C_VEL
LIN {X 0,Y 305.599,Z 341.044,A -85,B 0,C 180,E1 -15856.02,E2 -15856.02} C_VEL
LIN {X 0,Y 305.581,Z 341.044,A -85,B 0,C 180,E1 -15859.445,E2 -15859.445} C_VEL
LIN {X 0,Y 305.496,Z 341.054,A -85,B 0,C 180,E1 -15863.041,E2 -15863.041} C_VEL
LIN {X 0,Y 305.536,Z 341.048,A -85,B 0,C 180,E1 -15866.221,E2 -15866.221} C_VEL
LIN {X 0,Y 305.493,Z 341.054,A -85,B 0,C 180,E1 -15869.047,E2 -15869.047} C_VEL
LIN {X 0,Y 305.447,Z 341.061,A -85,B 0,C 180,E1 -15871.952,E2 -15871.952} C_VEL
LIN {X 0,Y 305.467,Z 341.06,A -85,B 0,C 180,E1 -15875.113,E2 -15875.113} C_VEL
LIN {X 0,Y 305.446,Z 341.055,A -85,B 0,C 180,E1 -15878.527,E2 -15878.527} C_VEL
LIN {X 0,Y 305.463,Z 341.058,A -85,B 0,C 180,E1 -15882.586,E2 -15882.586} C_VEL
LIN {X 0,Y 305.448,Z 341.059,A -85,B 0,C 180,E1 -15886.348,E2 -15886.348} C_VEL
LIN {X 0,Y 305.463,Z 341.059,A -85,B 0,C 180,E1 -15889.892,E2 -15889.892} C_VEL
LIN {X 0,Y 305.529,Z 341.242,A -85,B 0,C 180,E1 -15893.918,E2 -15893.918} C_VEL
LIN {X 0,Y 308.42,Z 353.733,A -85,B 0,C 180,E1 -15897.472,E2 -15897.472} C_VEL
LIN {X 0,Y 310.249,Z 362.284,A -85,B 0,C 180,E1 -15899.801,E2 -15899.801} C_VEL
LIN {X 0,Y 314.777,Z 374.552,A -85,B 0,C 180,E1 -15900.504,E2 -15900.504} C_VEL
LIN {X 0,Y 320.276,Z 410.699,A -85,B 0,C 180,E1 -15901.839,E2 -15901.839} C_VEL
LIN {X 0,Y 317.814,Z 500.638,A -85,B 0,C 180,E1 -15903.882,E2 -15903.882} C_VEL
LIN {X 0,Y 316.928,Z 515.343,A -85,B 0,C 180,E1 -15904.466,E2 -15904.466} C_VEL
LIN {X 0,Y 315.527,Z 529.94,A -85,B 0,C 180,E1 -15905.314,E2 -15905.314} C_VEL
LIN {X 0,Y 314.029,Z 543.264,A -85,B 0,C 180,E1 -15906.367,E2 -15906.367} C_VEL
LIN {X 0,Y 312.407,Z 556.234,A -85,B 0,C 180,E1 -15907.689,E2 -15907.689} C_VEL
LIN {X 0,Y 310.683,Z 567.605,A -85,B 0,C 180,E1 -15909.127,E2 -15909.127} C_VEL
LIN {X 0,Y 309.033,Z 578.069,A -85,B 0,C 180,E1 -15910.745,E2 -15910.745} C_VEL
LIN {X 0,Y 307.462,Z 588.465,A -85,B 0,C 180,E1 -15912.712,E2 -15912.712} C_VEL
LIN {X 0,Y 306.066,Z 597.588,A -85,B 0,C 180,E1 -15914.835,E2 -15914.835} C_VEL
LIN {X 0,Y 305.235,Z 604.196,A -85,B 0,C 180,E1 -15916.687,E2 -15916.687} C_VEL
LIN {X 0,Y 304.462,Z 610.084,A -85,B 0,C 180,E1 -15918.684,E2 -15918.684} C_VEL
LIN {X 0,Y 304.017,Z 614.924,A -85,B 0,C 180,E1 -15920.686,E2 -15920.686} C_VEL
LIN {X 0,Y 303.735,Z 619.912,A -85,B 0,C 180,E1 -15923.355,E2 -15923.355} C_VEL
LIN {X 0,Y 303.655,Z 623.359,A -85,B 0,C 180,E1 -15926.017,E2 -15926.017} C_VEL
LIN {X 0,Y 303.645,Z 625.374,A -85,B 0,C 180,E1 -15928.673,E2 -15928.673} C_VEL
LIN {X 0,Y 303.671,Z 625.864,A -85,B 0,C 180,E1 -15929.999,E2 -15929.999} C_VEL
LIN {X 0,Y 303.62,Z 625.822,A -85,B 0,C 180,E1 -15932.652,E2 -15932.652} C_VEL
LIN {X 0,Y 303.618,Z 624.436,A -85,B 0,C 180,E1 -15935.311,E2 -15935.311} C_VEL
LIN {X 0,Y 303.869,Z 621.695,A -85,B 0,C 180,E1 -15937.975,E2 -15937.975} C_VEL
LIN {X 0,Y 304.43,Z 617.536,A -85,B 0,C 180,E1 -15940.642,E2 -15940.642} C_VEL
LIN {X 0,Y 305.557,Z 611.846,A -85,B 0,C 180,E1 -15943.296,E2 -15943.296} C_VEL
LIN {X 0,Y 307.072,Z 604.465,A -85,B 0,C 180,E1 -15945.94,E2 -15945.94} C_VEL
LIN {X 0,Y 308.948,Z 596.367,A -85,B 0,C 180,E1 -15948.226,E2 -15948.226} C_VEL
LIN {X 0,Y 310.986,Z 587.923,A -85,B 0,C 180,E1 -15950.158,E2 -15950.158} C_VEL
LIN {X 0,Y 313.431,Z 577.782,A -85,B 0,C 180,E1 -15952.059,E2 -15952.059} C_VEL
LIN {X 0,Y 315.685,Z 567.62,A -85,B 0,C 180,E1 -15953.622,E2 -15953.622} C_VEL
LIN {X 0,Y 318.087,Z 555.564,A -85,B 0,C 180,E1 -15955.134,E2 -15955.134} C_VEL
LIN {X 0,Y 320.362,Z 543.099,A -85,B 0,C 180,E1 -15956.373,E2 -15956.373} C_VEL
LIN {X 0,Y 322.438,Z 529.603,A -85,B 0,C 180,E1 -15957.415,E2 -15957.415} C_VEL
LIN {X 0,Y 324.19,Z 515.493,A -85,B 0,C 180,E1 -15958.219,E2 -15958.219} C_VEL
LIN {X 0,Y 325.424,Z 501.673,A -85,B 0,C 180,E1 -15958.762,E2 -15958.762} C_VEL
LIN {X 0,Y 326.53,Z 474.896,A -85,B 0,C 180,E1 -15959.405,E2 -15959.405} C_VEL
LIN {X 0,Y 328.664,Z 412.182,A -85,B 0,C 180,E1 -15960.824,E2 -15960.824} C_VEL
LIN {X 0,Y 325.841,Z 395.107,A -85,B 0,C 180,E1 -15961.647,E2 -15961.647} C_VEL
LIN {X 0,Y 324.368,Z 387.981,A -85,B 0,C 180,E1 -15962.036,E2 -15962.036} C_VEL
LIN {X 0,Y 317.56,Z 373.437,A -85,B 0,C 180,E1 -15963.379,E2 -15963.379} C_VEL
LIN {X 0,Y 312.657,Z 364.129,A -85,B 0,C 180,E1 -15964.374,E2 -15964.374} C_VEL
LIN {X 0,Y 311.088,Z 360.81,A -85,B 0,C 180,E1 -15964.736,E2 -15964.736} C_VEL
LIN {X 0,Y 308.225,Z 350.287,A -85,B 0,C 180,E1 -15968.343,E2 -15968.343} C_VEL
LIN {X 0,Y 305.481,Z 341.046,A -85,B 0,C 180,E1 -15971.848,E2 -15971.848} C_VEL
LIN {X 0,Y 305.399,Z 341.052,A -85,B 0,C 180,E1 -15975.509,E2 -15975.509} C_VEL
LIN {X 0,Y 305.436,Z 341.066,A -85,B 0,C 180,E1 -15978.142,E2 -15978.142} C_VEL
LIN {X 0,Y 305.49,Z 341.044,A -85,B 0,C 180,E1 -15981.599,E2 -15981.599} C_VEL
LIN {X 0,Y 305.457,Z 341.058,A -85,B 0,C 180,E1 -15984.886,E2 -15984.886} C_VEL
LIN {X 0,Y 305.447,Z 341.062,A -85,B 0,C 180,E1 -15988.354,E2 -15988.354} C_VEL
LIN {X 0,Y 305.515,Z 341.051,A -85,B 0,C 180,E1 -15991.113,E2 -15991.113} C_VEL
LIN {X 0,Y 305.565,Z 341.04,A -85,B 0,C 180,E1 -15994.087,E2 -15994.087} C_VEL
LIN {X 0,Y 305.493,Z 341.054,A -85,B 0,C 180,E1 -15998.402,E2 -15998.402} C_VEL
LIN {X 0,Y 305.583,Z 341.035,A -85,B 0,C 180,E1 -16001.217,E2 -16001.217} C_VEL
LIN {X 0,Y 305.642,Z 341.028,A -85,B 0,C 180,E1 -16005.348,E2 -16005.348} C_VEL
LIN {X 0,Y 305.63,Z 341.029,A -85,B 0,C 180,E1 -16009.399,E2 -16009.399} C_VEL
LIN {X 0,Y 305.804,Z 341.012,A -85,B 0,C 180,E1 -16012.074,E2 -16012.074} C_VEL
LIN {X 0,Y 305.671,Z 341.034,A -85,B 0,C 180,E1 -16014.723,E2 -16014.723} C_VEL
LIN {X 0,Y 305.94,Z 341,A -85,B 0,C 180,E1 -16018.683,E2 -16018.683} C_VEL
LIN {X 0,Y 305.927,Z 340.993,A -85,B 0,C 180,E1 -16021.316,E2 -16021.316} C_VEL
LIN {X 0,Y 305.651,Z 341.028,A -85,B 0,C 180,E1 -16025.277,E2 -16025.277} C_VEL
LIN {X 0,Y 305.736,Z 341.023,A -85,B 0,C 180,E1 -16027.927,E2 -16027.927} C_VEL
LIN {X 0,Y 305.588,Z 341.039,A -85,B 0,C 180,E1 -16031.945,E2 -16031.945} C_VEL
LIN {X 0,Y 305.599,Z 341.043,A -85,B 0,C 180,E1 -16035.014,E2 -16035.014} C_VEL
LIN {X 0,Y 305.508,Z 341.051,A -85,B 0,C 180,E1 -16038.787,E2 -16038.787} C_VEL
LIN {X 0,Y 305.477,Z 341.055,A -85,B 0,C 180,E1 -16043.039,E2 -16043.039} C_VEL
LIN {X 0,Y 305.46,Z 341.063,A -85,B 0,C 180,E1 -16046.197,E2 -16046.197} C_VEL
LIN {X 0,Y 305.439,Z 341.047,A -85,B 0,C 180,E1 -16049.034,E2 -16049.034} C_VEL
LIN {X 0,Y 305.428,Z 341.061,A -85,B 0,C 180,E1 -16051.953,E2 -16051.953} C_VEL
LIN {X 0,Y 305.503,Z 341.236,A -85,B 0,C 180,E1 -16055.534,E2 -16055.534} C_VEL
LIN {X 0,Y 306.272,Z 343.877,A -85,B 0,C 180,E1 -16056.567,E2 -16056.567} C_VEL
LIN {X 0,Y 315.734,Z 359.703,A -85,B 0,C 180,E1 -16058.52,E2 -16058.52} C_VEL
LIN {X 0,Y 323.678,Z 374.593,A -85,B 0,C 180,E1 -16060.067,E2 -16060.067} C_VEL
LIN {X 0,Y 329.586,Z 387.33,A -85,B 0,C 180,E1 -16061.188,E2 -16061.188} C_VEL
LIN {X 0,Y 326.107,Z 479.742,A -85,B 0,C 180,E1 -16063.285,E2 -16063.285} C_VEL
LIN {X 0,Y 325.099,Z 493.677,A -85,B 0,C 180,E1 -16063.838,E2 -16063.838} C_VEL
LIN {X 0,Y 323.708,Z 506.663,A -85,B 0,C 180,E1 -16064.572,E2 -16064.572} C_VEL
LIN {X 0,Y 322.128,Z 518.983,A -85,B 0,C 180,E1 -16065.504,E2 -16065.504} C_VEL
LIN {X 0,Y 320.249,Z 530.673,A -85,B 0,C 180,E1 -16066.615,E2 -16066.615} C_VEL
LIN {X 0,Y 317.962,Z 542.704,A -85,B 0,C 180,E1 -16068.041,E2 -16068.041} C_VEL
LIN {X 0,Y 315.471,Z 554.333,A -85,B 0,C 180,E1 -16069.757,E2 -16069.757} C_VEL
LIN {X 0,Y 313.246,Z 564.227,A -85,B 0,C 180,E1 -16071.565,E2 -16071.565} C_VEL
LIN {X 0,Y 310.961,Z 573.417,A -85,B 0,C 180,E1 -16073.612,E2 -16073.612} C_VEL
LIN {X 0,Y 308.985,Z 581.157,A -85,B 0,C 180,E1 -16075.742,E2 -16075.742} C_VEL
LIN {X 0,Y 307.167,Z 588.413,A -85,B 0,C 180,E1 -16078.25,E2 -16078.25} C_VEL
LIN {X 0,Y 305.713,Z 594.197,A -85,B 0,C 180,E1 -16080.876,E2 -16080.876} C_VEL
LIN {X 0,Y 304.789,Z 598.144,A -85,B 0,C 180,E1 -16083.281,E2 -16083.281} C_VEL
LIN {X 0,Y 304.144,Z 600.67,A -85,B 0,C 180,E1 -16085.423,E2 -16085.423} C_VEL
LIN {X 0,Y 303.751,Z 602.372,A -85,B 0,C 180,E1 -16087.742,E2 -16087.742} C_VEL
LIN {X 0,Y 303.52,Z 603.047,A -85,B 0,C 180,E1 -16089.678,E2 -16089.678} C_VEL
LIN {X 0,Y 303.422,Z 602.781,A -85,B 0,C 180,E1 -16092.477,E2 -16092.477} C_VEL
LIN {X 0,Y 303.476,Z 601.091,A -85,B 0,C 180,E1 -16095.243,E2 -16095.243} C_VEL
LIN {X 0,Y 303.883,Z 597.959,A -85,B 0,C 180,E1 -16097.988,E2 -16097.988} C_VEL
LIN {X 0,Y 304.422,Z 593.339,A -85,B 0,C 180,E1 -16100.701,E2 -16100.701} C_VEL
LIN {X 0,Y 305.117,Z 588.382,A -85,B 0,C 180,E1 -16102.872,E2 -16102.872} C_VEL
LIN {X 0,Y 306.107,Z 581.104,A -85,B 0,C 180,E1 -16105.392,E2 -16105.392} C_VEL
LIN {X 0,Y 307.424,Z 572.618,A -85,B 0,C 180,E1 -16107.708,E2 -16107.708} C_VEL
LIN {X 0,Y 308.876,Z 563.758,A -85,B 0,C 180,E1 -16109.675,E2 -16109.675} C_VEL
LIN {X 0,Y 310.437,Z 553.072,A -85,B 0,C 180,E1 -16111.623,E2 -16111.623} C_VEL
LIN {X 0,Y 312.125,Z 542.212,A -85,B 0,C 180,E1 -16113.228,E2 -16113.228} C_VEL
LIN {X 0,Y 313.709,Z 530.369,A -85,B 0,C 180,E1 -16114.659,E2 -16114.659} C_VEL
LIN {X 0,Y 315.263,Z 517.297,A -85,B 0,C 180,E1 -16115.919,E2 -16115.919} C_VEL
